	            IF #i_boFinishedOk OR #i_boErr THEN
	                #io_stTask1.bo_InProgress := FALSE;
	                #io_boAnyInProgress := FALSE;
	                #io_boEnable := FALSE;
	            END_IF;
	            
	        ELSIF #io_stTask2.bo_InProgress THEN
	            IF #i_boFinishedOk THEN
	                #io_stTask2.bo_FinishedOk := TRUE;
	            END_IF;
	            IF #i_boErr THEN
	                #io_stTask2.bo_FinishedError := TRUE;
	            END_IF;
	            
	            IF #i_boFinishedOk OR #i_boErr THEN
	                #io_stTask2.bo_InProgress := FALSE;
	                #io_boAnyInProgress := FALSE;
	                #io_boEnable := FALSE;
	            END_IF;
	            
	        ELSIF #io_stTask3.bo_InProgress THEN
	            IF #i_boFinishedOk THEN
	                #io_stTask3.bo_FinishedOk := TRUE;
	            END_IF;
	            IF #i_boErr THEN
	                #io_stTask3.bo_FinishedError := TRUE;
	            END_IF;
	            
	            IF #i_boFinishedOk OR #i_boErr THEN
	                #io_stTask3.bo_InProgress := FALSE;
	                #io_boAnyInProgress := FALSE;
	                #io_boEnable := FALSE;
	            END_IF;
	        END_IF;
	    END_IF;
	    
	    // 3. Запуск новой задачи из очереди (по приоритету 1 -> 2 -> 3)
	    IF NOT #io_boAnyInProgress AND NOT #io_boEnable THEN
	        IF #io_stTask1.bo_Trigger THEN
	            #io_iCmdInput := #io_stTask1.i_Code;
	            #io_stTask1.bo_InProgress := TRUE;
	            #io_boAnyInProgress := TRUE;
	            #io_boEnable := TRUE;
	            #io_stTask1.bo_Trigger := FALSE;
	            
	        ELSIF #io_stTask2.bo_Trigger THEN
	            #io_iCmdInput := #io_stTask2.i_Code;
	            #io_stTask2.bo_InProgress := TRUE;
	            #io_boAnyInProgress := TRUE;
	            #io_boEnable := TRUE;
	            #io_stTask2.bo_Trigger := FALSE;
	            
	        ELSIF #io_stTask3.bo_Trigger THEN
	            #io_iCmdInput := #io_stTask3.i_Code;
	            #io_stTask3.bo_InProgress := TRUE;
	            #io_boAnyInProgress := TRUE;
	            #io_boEnable := TRUE;
	            #io_stTask3.bo_Trigger := FALSE;
	        END_IF;
	    END_IF;
END_FUNCTION

FUNCTION_BLOCK "FB_Map_Siwarex_Core"
TITLE = Маппинг данных Siwarex CS
{ S7_Optimized_Access := 'FALSE' }
AUTHOR : S7C_Lib
FAMILY : Analog
VERSION : 1.4
// ==============================================================================
// Описание: Адаптированный маппинг из UDT_SIWA_CS. Обработка раздельных кодов 
//           ошибок (модуля и драйвера). Встроенный таймер Watchdog в STAT.
// ==============================================================================
   VAR 
      stat_Diag_CS_1 { ExternalAccessible := 'False'; ExternalVisible := 'False'; ExternalWritable := 'False'} : Struct   // Внутренняя память для Watchdog
         Old_Count { ExternalAccessible := 'False'; ExternalVisible := 'False'; ExternalWritable := 'False'} : Byte;
         Old_Weight { ExternalAccessible := 'False'; ExternalVisible := 'False'; ExternalWritable := 'False'} : Real;
         Last_Change_ms { ExternalAccessible := 'False'; ExternalVisible := 'False'; ExternalWritable := 'False'} : Real;
      END_STRUCT;
      stat_Diag_CS_2 { ExternalAccessible := 'False'; ExternalVisible := 'False'; ExternalWritable := 'False'} : Struct   // Внутренняя память для Watchdog
         Old_Count { ExternalAccessible := 'False'; ExternalVisible := 'False'; ExternalWritable := 'False'} : Byte;
         Old_Weight { ExternalAccessible := 'False'; ExternalVisible := 'False'; ExternalWritable := 'False'} : Real;
         Last_Change_ms { ExternalAccessible := 'False'; ExternalVisible := 'False'; ExternalWritable := 'False'} : Real;
      END_STRUCT;
   END_VAR

   VAR_TEMP 
      temp_Value_Changed : Bool;
      temp_Counter_Changed : Bool;
   END_VAR


BEGIN
	
	// ============================================================================
	// SCALE CS_1
	// ============================================================================
	
	// 1. Веса
	"DB_MAP".Scale_CS_1.Weight_Gross_kg := INT_TO_REAL("DB_SCALE_CS_1".s_PROCESS_VALUES.i_GROSS_WEIGHT_PROC);
	"DB_MAP".Scale_CS_1.Weight_Net_kg := INT_TO_REAL("DB_SCALE_CS_1".s_PROCESS_VALUES.i_NET_WEIGHT_PROC);
	"DB_MAP".Scale_CS_1.Weight_Tare_kg := INT_TO_REAL("DB_SCALE_CS_1".s_PROCESS_VALUES.i_TARE_WEIGHT_PROC);
	
	// 2. Статусы
	"DB_MAP".Scale_CS_1.Status.Standstill := "DB_SCALE_CS_1".s_PROCESS_VALUES.bo_STA_ST_STAND_SCALE_ON;
	"DB_MAP".Scale_CS_1.Status.Limit_1 := "DB_SCALE_CS_1".s_PROCESS_VALUES.bo_STA_LIMIT1_ON;
	"DB_MAP".Scale_CS_1.Status.Limit_2 := "DB_SCALE_CS_1".s_PROCESS_VALUES.bo_STA_LIMIT2_ON;
	"DB_MAP".Scale_CS_1.Status.Tared := "DB_SCALE_CS_1".s_PROCESS_VALUES.bo_STA_TARED;
	"DB_MAP".Scale_CS_1.Status.Quarter_D_Zero := "DB_SCALE_CS_1".s_PROCESS_VALUES.bo_STA_025_D_ZERO;
	"DB_MAP".Scale_CS_1.Status.Scale_Calibrated := "DB_SCALE_CS_1".s_PROCESS_VALUES.bo_STA_SCALE_CALIBRATED;
	"DB_MAP".Scale_CS_1.Status.Write_Protected := "DB_SCALE_CS_1".s_PROCESS_VALUES.bo_STA_WRI_PROT;
	"DB_MAP".Scale_CS_1.Status.Limit_Max := "DB_SCALE_CS_1".s_PROCESS_VALUES.bo_STA_MAX_9E;
	"DB_MAP".Scale_CS_1.Status.Fault_HW := "DB_SCALE_CS_1".s_PROCESS_VALUES.bo_STA_ERROR_ON;
	"DB_MAP".Scale_CS_1.Status.Fault_FB := "DB_SCALE_CS_1".bo_FB_ERR;
	"DB_MAP".Scale_CS_1.Status.Fault := "DB_SCALE_CS_1".s_PROCESS_VALUES.bo_STA_ERROR_ON OR "DB_SCALE_CS_1".bo_FB_ERR;
	
	// 3. Коды ошибок: старший байт = b_OPR_ERR_MSG, младший = b_FB_ERR_CODE
	"DB_MAP".Scale_CS_1.Err_Raw :=
	    SHL(IN := BYTE_TO_WORD("DB_SCALE_CS_1".s_PROCESS_VALUES.b_OPR_ERR_MSG), N := 8)
	    OR BYTE_TO_WORD("DB_SCALE_CS_1".b_FB_ERR_CODE);
	
	// 4. Watchdog CS_1
	#temp_Value_Changed := ("DB_MAP".Scale_CS_1.Weight_Net_kg <> #stat_Diag_CS_1.Old_Weight);
	#temp_Counter_Changed := ("DB_SCALE_CS_1".b_INFO_REFRESH_COUNT <> #stat_Diag_CS_1.Old_Count);
	
	IF #temp_Counter_Changed THEN //#temp_Value_Changed OR 
	    #stat_Diag_CS_1.Last_Change_ms := 0.0;
	    #stat_Diag_CS_1.Old_Weight := "DB_MAP".Scale_CS_1.Weight_Net_kg;
	    #stat_Diag_CS_1.Old_Count := "DB_SCALE_CS_1".b_INFO_REFRESH_COUNT;
	    "DB_MAP".Scale_CS_1.Status.Comm_Fault := FALSE;
	ELSE
	    #stat_Diag_CS_1.Last_Change_ms := #stat_Diag_CS_1.Last_Change_ms + "getCycleTime"();
	    IF #stat_Diag_CS_1.Last_Change_ms > 5000.0 THEN
	        "DB_MAP".Scale_CS_1.Status.Comm_Fault := TRUE;
	    END_IF;
	END_IF;
	
	
	// ============================================================================
	// SCALE CS_2
	// ============================================================================
	
	// 1. Веса
	"DB_MAP".Scale_CS_2.Weight_Gross_kg := INT_TO_REAL("DB_SCALE_CS_2".s_PROCESS_VALUES.i_GROSS_WEIGHT_PROC);
	"DB_MAP".Scale_CS_2.Weight_Net_kg := INT_TO_REAL("DB_SCALE_CS_2".s_PROCESS_VALUES.i_NET_WEIGHT_PROC);
	"DB_MAP".Scale_CS_2.Weight_Tare_kg := INT_TO_REAL("DB_SCALE_CS_2".s_PROCESS_VALUES.i_TARE_WEIGHT_PROC);
	
	// 2. Статусы
	"DB_MAP".Scale_CS_2.Status.Standstill := "DB_SCALE_CS_2".s_PROCESS_VALUES.bo_STA_ST_STAND_SCALE_ON;
	"DB_MAP".Scale_CS_2.Status.Limit_1 := "DB_SCALE_CS_2".s_PROCESS_VALUES.bo_STA_LIMIT1_ON;
	"DB_MAP".Scale_CS_2.Status.Limit_2 := "DB_SCALE_CS_2".s_PROCESS_VALUES.bo_STA_LIMIT2_ON;
	"DB_MAP".Scale_CS_2.Status.Tared := "DB_SCALE_CS_2".s_PROCESS_VALUES.bo_STA_TARED;
	"DB_MAP".Scale_CS_2.Status.Quarter_D_Zero := "DB_SCALE_CS_2".s_PROCESS_VALUES.bo_STA_025_D_ZERO;
	"DB_MAP".Scale_CS_2.Status.Scale_Calibrated := "DB_SCALE_CS_2".s_PROCESS_VALUES.bo_STA_SCALE_CALIBRATED;
	"DB_MAP".Scale_CS_2.Status.Write_Protected := "DB_SCALE_CS_2".s_PROCESS_VALUES.bo_STA_WRI_PROT;
	"DB_MAP".Scale_CS_2.Status.Limit_Max := "DB_SCALE_CS_2".s_PROCESS_VALUES.bo_STA_MAX_9E;
	"DB_MAP".Scale_CS_2.Status.Fault_HW := "DB_SCALE_CS_2".s_PROCESS_VALUES.bo_STA_ERROR_ON;
	"DB_MAP".Scale_CS_2.Status.Fault_FB := "DB_SCALE_CS_2".bo_FB_ERR;
	"DB_MAP".Scale_CS_2.Status.Fault := "DB_SCALE_CS_2".s_PROCESS_VALUES.bo_STA_ERROR_ON OR "DB_SCALE_CS_2".bo_FB_ERR;
	// 3. Коды ошибок
	"DB_MAP".Scale_CS_2.Err_Raw :=
	SHL(IN := BYTE_TO_WORD("DB_SCALE_CS_2".s_PROCESS_VALUES.b_OPR_ERR_MSG), N := 8)
	OR BYTE_TO_WORD("DB_SCALE_CS_2".b_FB_ERR_CODE);
	
	// 4. Watchdog CS_2
	#temp_Value_Changed := ("DB_MAP".Scale_CS_2.Weight_Net_kg <> #stat_Diag_CS_2.Old_Weight);
	#temp_Counter_Changed := ("DB_SCALE_CS_2".b_INFO_REFRESH_COUNT <> #stat_Diag_CS_2.Old_Count);
	
	IF #temp_Counter_Changed THEN //#temp_Value_Changed OR 
	    #stat_Diag_CS_2.Last_Change_ms := 0.0;
	    #stat_Diag_CS_2.Old_Weight := "DB_MAP".Scale_CS_2.Weight_Net_kg;
	    #stat_Diag_CS_2.Old_Count := "DB_SCALE_CS_2".b_INFO_REFRESH_COUNT;
	    "DB_MAP".Scale_CS_2.Status.Comm_Fault := FALSE;
	ELSE
	    #stat_Diag_CS_2.Last_Change_ms := #stat_Diag_CS_2.Last_Change_ms + "getCycleTime"();
	    IF #stat_Diag_CS_2.Last_Change_ms > 5000.0 THEN
	        "DB_MAP".Scale_CS_2.Status.Comm_Fault := TRUE;
	    END_IF;
	END_IF;
	
END_FUNCTION_BLOCK

FUNCTION "getCycleTime" : Real
{ S7_Optimized_Access := 'FALSE' }
VERSION : 0.1

BEGIN
	#getCycleTime := "DB_Global".Sys.CycleTime_ms_REAL;
END_FUNCTION

ORGANIZATION_BLOCK "COMPLETE RESTART"
TITLE = "Complete Restart"
{ S7_Optimized_Access := 'FALSE' }
VERSION : 0.1
   VAR_TEMP 
      OB100_EV_CLASS : Byte;   // 16#13, Event class 1, Entering event state, Event logged in diagnostic buffer
      OB100_STRTUP : Byte;   // 16#81/82/83/84 Method of startup
      OB100_PRIORITY : Byte;   // Priority of OB Execution
      OB100_OB_NUMBR : Byte;   // 100 (Organization block 100, OB100)
      OB100_RESERVED_1 : Byte;   // Reserved for system
      OB100_RESERVED_2 : Byte;   // Reserved for system
      OB100_STOP : Word;   // Event that caused CPU to stop (16#4xxx)
      OB100_STRT_INFO : DWord;   // Information on how system started
      OB100_DATE_TIME : Date_And_Time;   // Date and time OB100 started
   END_VAR


BEGIN
	"Total_DB".first_scan := TRUE;
	
END_ORGANIZATION_BLOCK

ORGANIZATION_BLOCK "CYC_INT5"
TITLE = "Cyclic Interrupt"
{ S7_Optimized_Access := 'FALSE' }
VERSION : 0.1
   VAR_TEMP 
      OB35_EV_CLASS : Byte;   // Bits 0-3 = 1 (Coming event), Bits 4-7 = 1 (Event class 1)
      OB35_STRT_INF : Byte;   // 16#36 (OB 35 has started)
      OB35_PRIORITY : Byte;   // Priority of OB Execution
      OB35_OB_NUMBR : Byte;   // 35 (Organization block 35, OB35)
      OB35_RESERVED_1 : Byte;   // Reserved for system
      OB35_RESERVED_2 : Byte;   // Reserved for system
      OB35_PHASE_OFFSET : Word;   // Phase offset (msec)
      OB35_RESERVED_3 : Int;   // Reserved for system
      OB35_EXC_FREQ : Int;   // Frequency of execution (msec)
      OB35_DATE_TIME : Date_And_Time;   // Date and time OB35 started
   END_VAR


BEGIN
	// Опрос Танка 1 (Слот 3 - фоновое чтение веса)
	"FC_Weighing_Poll"(
	                   i_boAnyInProgress := "DB_SCALE_CS_1".bo_CMD_IN_PROGRESS,
	                   i_boCmdEnable     := "DB_SCALE_CS_1".bo_CMD_TRIGGER,
	                   io_stTask          := "DB_SCALE_CS_1".s_CMD3
	);
	
	// Опрос Танка 2 (Слот 3 - фоновое чтение веса)
	"FC_Weighing_Poll"(
	                   i_boAnyInProgress := "DB_SCALE_CS_2".bo_CMD_IN_PROGRESS,
	                   i_boCmdEnable     := "DB_SCALE_CS_2".bo_CMD_TRIGGER,
	                   io_stTask          := "DB_SCALE_CS_2".s_CMD3
	);
END_ORGANIZATION_BLOCK

FUNCTION "FC_Weighing_Poll" : Void
{ S7_Optimized_Access := 'FALSE' }
VERSION : 1.2
   VAR_INPUT 
      i_boAnyInProgress : Bool;   // Общий статус занятости модуля
      i_boCmdEnable : Bool;   // Общий триггер команд модуля
   END_VAR

   VAR_IN_OUT 
      io_stTask : "UDT_SIWA_Cmd";   // Слот задачи циклического опроса (напр. sTask3)
   END_VAR


BEGIN
	    // ===================================================
	    // Генерация команды чтения Data Record (DR30 - Код 230)
	    // Функция предназначена для циклического вызова (OB35)
	    // ===================================================
	    IF NOT #i_boAnyInProgress AND NOT #i_boCmdEnable AND NOT #io_stTask.bo_InProgress THEN
	        #io_stTask.i_Code := 230;
	        #io_stTask.bo_Trigger := TRUE;
	    END_IF;
	    
END_FUNCTION

FUNCTION_BLOCK "FB_AI"
TITLE = Functional block from AI
{ S7_Optimized_Access := 'FALSE' }
AUTHOR : Gemini
FAMILY : Arhive
VERSION : 8.0
// -----------------------------------------------------------------------------
// БЛОК ОБРАБОТКИ АНАЛОГОВОГО СИГНАЛА (FB_AI)
// -----------------------------------------------------------------------------
   VAR_INPUT 
      i_iRawSignal : Int;
      i_rSimValue : Real;
   END_VAR

   VAR_IN_OUT 
      io_stConfig : "UDT_AI_Conf";
      io_stOut : "UDT_AI_Out";
   END_VAR

   VAR 
      stat_boWasInvalid : Bool := TRUE;
   END_VAR

   VAR_TEMP 
      temp_boDisabled : Bool;
      temp_boSimActive : Bool;
      temp_boUseSqrt : Bool;
      temp_boPreSqrtCut : Bool;
      temp_boFinalClamp : Bool;
      temp_rMA : Real;
      temp_rNorm : Real;
      temp_rCutoff_Norm : Real;
      temp_rScaled : Real;
      temp_rRange_mA : Real;
      temp_rRange_Phys : Real;
      temp_rMinPhys : Real;
      temp_rMaxPhys : Real;
      temp_boResetFilter : Bool;
      temp_iFilterTime : Int;
   END_VAR


BEGIN
	    // =========================================================
	    // ШАГ 0. РАСШИФРОВКА БИТОВОГО СЛОВА (Mode)
	    // =========================================================
	    #temp_boDisabled := (#io_stConfig.Mode AND 16#0001) = 16#0001;
	    #temp_boSimActive := (#io_stConfig.Mode AND 16#0002) = 16#0002;
	    #temp_boUseSqrt := (#io_stConfig.Mode AND 16#0004) = 16#0004;
	    #temp_boPreSqrtCut := (#io_stConfig.Mode AND 16#0008) = 16#0008;
	    #temp_boFinalClamp := (#io_stConfig.Mode AND 16#0010) = 16#0010;
	    
	    // 0.1 Режим полного отключения канала
	    IF #temp_boDisabled THEN
	        #io_stOut.Value_Unclamped := 0.0;
	        #io_stOut.Value_Scaled := 0.0;
	        #io_stOut.Value_Filtered := 0.0;
	        #io_stOut.Value_mA := 0.0;
	        #io_stOut.Raw := 0;
	        
	        #io_stOut.Status.WireBreak := FALSE;
	        #io_stOut.Status.Underrange := FALSE;
	        #io_stOut.Status.Overrange := FALSE;
	        #io_stOut.Status.Overflow := FALSE;
	        #io_stOut.Status.ConfigError := FALSE;
	        #io_stOut.Status.Sim_Active := FALSE;
	        
	        #stat_boWasInvalid := TRUE;
	        RETURN;
	    END_IF;
	    
	    // 0.2 Защита от ошибок конфигурации
	    #temp_rRange_mA := #io_stConfig.Calib_mA_Max - #io_stConfig.Calib_mA_Min;
	    #temp_rRange_Phys := #io_stConfig.Scale_Max - #io_stConfig.Scale_Min;
	    
	    IF (#io_stConfig.HW_Max <= #io_stConfig.HW_Min) OR
	        (#temp_rRange_mA <= 0.0) OR
	        (ABS(#temp_rRange_Phys) < 0.00001) OR
	        (ABS(#io_stConfig.Cutoff) >= ABS(#temp_rRange_Phys)) THEN
	        
	        #io_stOut.Status.ConfigError := TRUE;
	        
	        #io_stOut.Status.WireBreak := FALSE;
	        #io_stOut.Status.Underrange := FALSE;
	        #io_stOut.Status.Overrange := FALSE;
	        #io_stOut.Status.Overflow := FALSE;
	        #io_stOut.Status.Sim_Active := FALSE;
	        
	        #io_stOut.Value_Unclamped := 0.0;
	        #io_stOut.Value_Scaled := 0.0;
	        #io_stOut.Value_Filtered := 0.0;
	        #io_stOut.Value_mA := 0.0;
	        #io_stOut.Raw := #i_iRawSignal;
	        
	        #stat_boWasInvalid := TRUE;
	        RETURN;
	    END_IF;
	    
	    #io_stOut.Status.ConfigError := FALSE;
	    
	    // =========================================================
	    // ШАГ 1 & 2. СИМУЛЯЦИЯ И ДИАГНОСТИКА
	    // =========================================================
	    IF #temp_boSimActive THEN
	        #io_stOut.Status.Sim_Active := TRUE;
	        
	        #io_stOut.Status.WireBreak := FALSE;
	        #io_stOut.Status.Underrange := FALSE;
	        #io_stOut.Status.Overrange := FALSE;
	        #io_stOut.Status.Overflow := FALSE;
	        
	        #io_stOut.Raw := 0;
	        #io_stOut.Value_mA := 0.0;
	        #temp_rScaled := #i_rSimValue;
	    ELSE
	        #io_stOut.Status.Sim_Active := FALSE;
	        #io_stOut.Raw := #i_iRawSignal;
	        
	        "FC_AnalogDiag"(
	                        i_iRawSignal := #i_iRawSignal,
	                        i_iHW_Min := #io_stConfig.HW_Min,
	                        i_iHW_Max := #io_stConfig.HW_Max,
	                        i_rCoef_Under := "C_DIAG_UNDER",
	                        i_rCoef_Over := "C_DIAG_OVER",
	                        o_boWireBreak => #io_stOut.Status.WireBreak,
	                        o_boUnderrange => #io_stOut.Status.Underrange,
	                        o_boOverrange => #io_stOut.Status.Overrange,
	                        o_boOverflow => #io_stOut.Status.Overflow
	        );
	        
	        // =========================================================
	        // ШАГ 3. МАТЕМАТИКА
	        // =========================================================
	        IF #io_stOut.Status.WireBreak THEN
	            #temp_rScaled := #io_stConfig.Scale_Min + (#temp_rRange_Phys * "C_DIAG_UNDER");
	            #io_stOut.Value_mA := 0.0;
	            
	        ELSIF #io_stOut.Status.Overflow THEN
	            #temp_rScaled := #io_stConfig.Scale_Min + (#temp_rRange_Phys * "C_DIAG_OVER");
	            #io_stOut.Value_mA := 25.0;
	            
	        ELSE
	            // А) Расчет миллиампер
	            #temp_rMA := 4.0 + ((INT_TO_REAL(#i_iRawSignal) - INT_TO_REAL(#io_stConfig.HW_Min)) /
	            (INT_TO_REAL(#io_stConfig.HW_Max) - INT_TO_REAL(#io_stConfig.HW_Min))) * 16.0;
	            #io_stOut.Value_mA := #temp_rMA;
	            
	            // Б) Нормализация (0.0 ... 1.0)
	            #temp_rNorm := (#temp_rMA - #io_stConfig.Calib_mA_Min) / #temp_rRange_mA;
	            
	            // В & Г) Работа с корнем (Отсечка и извлечение)
	            IF #temp_boUseSqrt THEN
	                
	                IF #temp_boPreSqrtCut THEN
	                    #temp_rCutoff_Norm := #io_stConfig.Cutoff / #temp_rRange_Phys;
	                    #temp_rCutoff_Norm := #temp_rCutoff_Norm * #temp_rCutoff_Norm;
	                    
	                    IF #temp_rNorm < #temp_rCutoff_Norm THEN
	                        #temp_rNorm := 0.0;
	                    END_IF;
	                END_IF;
	                
	                IF #temp_rNorm > 0.0 THEN
	                    #temp_rNorm := SQRT(#temp_rNorm);
	                ELSE
	                    #temp_rNorm := 0.0;
	                END_IF;
	                
	            END_IF;
	            
	            // Д) Масштабирование в физическую величину
	            #temp_rScaled := #io_stConfig.Scale_Min + (#temp_rNorm * #temp_rRange_Phys);
	            
	            // Е) Классический CutOff (только если не применялся Pre-Sqrt)
	            IF NOT (#temp_boPreSqrtCut AND #temp_boUseSqrt) THEN
	                IF ABS(#temp_rScaled) < ABS(#io_stConfig.Cutoff) THEN
	                    #temp_rScaled := 0.0;
	                END_IF;
	            END_IF;
	        END_IF;
	    END_IF;
	    
	    // Сохраняем чистую математику на выход
	    #io_stOut.Value_Unclamped := #temp_rScaled;
	    
	    // =========================================================
	    // ШАГ 3.5. ФИНАЛЬНЫЙ CLAMP
	    // =========================================================
	    IF #temp_boFinalClamp THEN
	        #temp_rMinPhys := MIN(IN1 := #io_stConfig.Scale_Min, IN2 := #io_stConfig.Scale_Max);
	        #temp_rMaxPhys := MAX(IN1 := #io_stConfig.Scale_Min, IN2 := #io_stConfig.Scale_Max);
	        #temp_rScaled := LIMIT(MN := #temp_rMinPhys, IN := #temp_rScaled, MX := #temp_rMaxPhys);
	    END_IF;
	    
	    #io_stOut.Value_Scaled := #temp_rScaled;
	    
	    // =========================================================
	    // ШАГ 4. ФИЛЬТРАЦИЯ & PRE-LOAD 
	    // =========================================================
	    #temp_boResetFilter := #temp_boSimActive OR
	    #io_stOut.Status.WireBreak OR
	    #io_stOut.Status.Overflow OR
	    #stat_boWasInvalid;
	    
	    #temp_iFilterTime := LIMIT(MN := 0, IN := #io_stConfig.FilterTime_ms, MX := 32000);
	    
	    "FC_Filter_PT1"(
	                    i_rRawValue := #temp_rScaled,
	                    i_rTimeFilter_ms := INT_TO_REAL(#temp_iFilterTime),
	                    i_boReset := #temp_boResetFilter,
	                    io_rFilteredValue := #io_stOut.Value_Filtered
	    );
	    
	    #stat_boWasInvalid := #io_stOut.Status.WireBreak OR
	    #io_stOut.Status.Overflow OR
	    #io_stOut.Status.ConfigError;
	    
END_FUNCTION_BLOCK

FUNCTION "FC_AnalogDiag" : Void
{ S7_Optimized_Access := 'FALSE' }
VERSION : 1.1
   VAR_INPUT 
      i_iRawSignal : Int;
      i_iHW_Min : Int;
      i_iHW_Max : Int;
      i_rCoef_Under : Real;
      i_rCoef_Over : Real;
   END_VAR

   VAR_OUTPUT 
      o_boWireBreak : Bool;
      o_boUnderrange : Bool;
      o_boOverrange : Bool;
      o_boOverflow : Bool;
   END_VAR

   VAR_TEMP 
      temp_iLimit_Max : Real;
      temp_iLimit_Min : Int;
      temp_rHWRange : Real;
   END_VAR


BEGIN
	#temp_rHWRange := INT_TO_REAL(#i_iHW_Max) - INT_TO_REAL(#i_iHW_Min);
	
	#temp_iLimit_Max := REAL_TO_INT(INT_TO_REAL(#i_iHW_Max) + (#i_rCoef_Over * #temp_rHWRange));
	#temp_iLimit_Min := REAL_TO_INT(INT_TO_REAL(#i_iHW_Min) + (#i_rCoef_Under * #temp_rHWRange));
	
	#o_boWireBreak := #i_iRawSignal < #temp_iLimit_Min;
	#o_boUnderrange := (#i_iRawSignal < #i_iHW_Min) AND (#i_iRawSignal >= #temp_iLimit_Min);
	#o_boOverrange := (#i_iRawSignal > #i_iHW_Max) AND (#i_iRawSignal <= #temp_iLimit_Max);
	#o_boOverflow := #i_iRawSignal >#temp_iLimit_Max;
END_FUNCTION

FUNCTION "FC_Filter_PT1" : Void
{ S7_Optimized_Access := 'FALSE' }
VERSION : 1.3
// ==========================================
// МАТЕМАТИКА: ФИЛЬТР ЭКСПОНЕНЦИАЛЬНОГО СГЛАЖИВАНИЯ (PT1)
// ==========================================
   VAR_INPUT 
      i_rRawValue : Real;
      i_rTimeFilter_ms : Real;
      i_boReset : Bool;
   END_VAR

   VAR_IN_OUT 
      io_rFilteredValue : Real;
   END_VAR

   VAR_TEMP 
      temp_rCycleTime_ms : Real;
      temp_rAlpha : Real;
   END_VAR


BEGIN
	#temp_rCycleTime_ms := "getCycleTime"();
	
	//Защита
	// -Ресет фильтра
	// -Защита от системного сбоя (если ПЛК выдал dt <= 0)
	// -Умный Safe State (по правилу Найквиста)
	//    Если заданное время фильтра меньше половины цикла ПЛК,
	//    фильтрация физически невозможна. Просто пробрасываем сигнал напрямую.
	IF #i_boReset OR #temp_rCycleTime_ms <= 0.000001 OR #i_rTimeFilter_ms < (#temp_rCycleTime_ms / 2.0) THEN
	    #io_rFilteredValue := #i_rRawValue;
	    RETURN;
	END_IF;
	
	IF #i_rTimeFilter_ms < 50.0 THEN
	    #temp_rAlpha := 1.0;
	    #io_rFilteredValue := #i_rRawValue;
	    RETURN;
	END_IF;
	
	
	// 3. Математика PT1
	#temp_rAlpha := #temp_rCycleTime_ms / (#i_rTimeFilter_ms + #temp_rCycleTime_ms);
	#io_rFilteredValue := #io_rFilteredValue + #temp_rAlpha * (#i_rRawValue - #io_rFilteredValue);
	
END_FUNCTION

FUNCTION_BLOCK "FB_AI_Alarm"
{ S7_Optimized_Access := 'FALSE' }
VERSION : 2.0
   VAR_INPUT 
      i_rValue : Real;
      i_boReset : Bool;
      i_boInhibit : Bool;
   END_VAR

   VAR_IN_OUT 
      io_stConfig : "UDT_AI_Alarm_Conf";
      io_stOut : "UDT_AI_Alarm";
   END_VAR

   VAR 
      stat_TonHiHi {InstructionName := 'TON'; LibVersion := '1.0'; S7_SetPoint := 'False'} : TON;
      stat_TonHi {InstructionName := 'TON'; LibVersion := '1.0'; S7_SetPoint := 'False'} : TON;
      stat_TonLo {InstructionName := 'TON'; LibVersion := '1.0'; S7_SetPoint := 'False'} : TON;
      stat_TonLoLo {InstructionName := 'TON'; LibVersion := '1.0'; S7_SetPoint := 'False'} : TON;
      stat_RawHiHi : Bool;
      stat_RawHi : Bool;
      stat_RawLo : Bool;
      stat_RawLoLo : Bool;
   END_VAR


BEGIN
	    // =========================================================
	    // 0. ЗАЩИТА ОТ ДУРАКА (Ограничение уставок времени >= 0)
	    // =========================================================
	    IF #io_stConfig.Delay_HiHi < 0 THEN
	        #io_stConfig.Delay_HiHi := 0;
	    END_IF;
	    IF #io_stConfig.Delay_Hi < 0 THEN
	        #io_stConfig.Delay_Hi := 0;
	    END_IF;
	    IF #io_stConfig.Delay_Lo < 0 THEN
	        #io_stConfig.Delay_Lo := 0;
	    END_IF;
	    IF #io_stConfig.Delay_LoLo < 0 THEN
	        #io_stConfig.Delay_LoLo := 0;
	    END_IF;
	    
	    // =========================================================
	    // 1. ТРАНСЛЯЦИЯ СТАТУСОВ ДЛЯ HMI (En_Out)
	    // =========================================================
	    #io_stOut.En_HiHi := #io_stConfig.En_Alarm.HiHi AND NOT #i_boInhibit;
	    #io_stOut.En_Hi := #io_stConfig.En_Alarm.Hi AND NOT #i_boInhibit;
	    #io_stOut.En_Lo := #io_stConfig.En_Alarm.Lo AND NOT #i_boInhibit;
	    #io_stOut.En_LoLo := #io_stConfig.En_Alarm.LoLo AND NOT #i_boInhibit;
	    #io_stOut.En_Latch_Enable := #io_stConfig.En_Alarm.Latch_Enable;
	    
	    // =========================================================
	    // 2. ОБРАБОТКА СЫРЫХ АВАРИЙ С ГИСТЕРЕЗИСОМ (Deadband)
	    // =========================================================
	    // Верхние пороги (Срабатывание >, Сброс <)
	    IF #i_rValue > #io_stConfig.HiHi THEN
	        #stat_RawHiHi := TRUE;
	    ELSIF #i_rValue < (#io_stConfig.HiHi - #io_stConfig.Hysteresis) THEN
	        #stat_RawHiHi := FALSE;
	    END_IF;
	    
	    IF #i_rValue > #io_stConfig.Hi THEN
	        #stat_RawHi := TRUE;
	    ELSIF #i_rValue < (#io_stConfig.Hi - #io_stConfig.Hysteresis) THEN
	        #stat_RawHi := FALSE;
	    END_IF;
	    
	    // Нижние пороги (Срабатывание <, Сброс >)
	    IF #i_rValue < #io_stConfig.Lo THEN
	        #stat_RawLo := TRUE;
	    ELSIF #i_rValue > (#io_stConfig.Lo + #io_stConfig.Hysteresis) THEN
	        #stat_RawLo := FALSE;
	    END_IF;
	    
	    IF #i_rValue < #io_stConfig.LoLo THEN
	        #stat_RawLoLo := TRUE;
	    ELSIF #i_rValue > (#io_stConfig.LoLo + #io_stConfig.Hysteresis) THEN
	        #stat_RawLoLo := FALSE;
	    END_IF;
	    
	    // =========================================================
	    // 3. ТАЙМЕРЫ ЗАДЕРЖКИ (ON-Delay)
	    // =========================================================
	    // Таймер не считает, если сработала блокировка датчика (Inhibit) 
	    // или аларм выключен в настройках.
	    #stat_TonHiHi(IN := #stat_RawHiHi AND #io_stConfig.En_Alarm.HiHi AND NOT #i_boInhibit,
	                  PT := DINT_TO_TIME(#io_stConfig.Delay_HiHi) * 1000 + t#1ms);//gr-ny 300
	    
	    #stat_TonHi(IN := #stat_RawHi AND #io_stConfig.En_Alarm.Hi AND NOT #i_boInhibit,
	                PT := DINT_TO_TIME(#io_stConfig.Delay_Hi) * 1000 + t#1ms);//gr-ny 300
	    
	    #stat_TonLo(IN := #stat_RawLo AND #io_stConfig.En_Alarm.Lo AND NOT #i_boInhibit,
	                PT := DINT_TO_TIME(#io_stConfig.Delay_Lo) * 1000 + t#1ms);//gr-ny 300
	    
	    #stat_TonLoLo(IN := #stat_RawLoLo AND #io_stConfig.En_Alarm.LoLo AND NOT #i_boInhibit,
	                  PT := DINT_TO_TIME(#io_stConfig.Delay_LoLo) * 1000 + t#1ms);//gr-ny 300
	    
	    // =========================================================
	    // 4. ФИКСАЦИЯ (LATCH) И СБРОС АВАРИЙ
	    // =========================================================
	    // Логика сброса (имеет приоритет):
	    // 1. Сработал Inhibit (глушим всё безусловно)
	    // 2. Аларм сняли в настройках
	    // 3. Уровень в норме И (нет фиксации ИЛИ нажата кнопка Reset)
	    
	    // --- HiHi ---
	    IF #i_boInhibit OR NOT #io_stConfig.En_Alarm.HiHi OR
	        (NOT #stat_RawHiHi AND (NOT #io_stConfig.En_Alarm.Latch_Enable OR #i_boReset)) THEN
	        #io_stOut.HiHi := FALSE;
	    ELSIF #stat_TonHiHi.Q THEN
	        #io_stOut.HiHi := TRUE;
	    END_IF;
	    
	    // --- Hi ---
	    IF #i_boInhibit OR NOT #io_stConfig.En_Alarm.Hi OR
	        (NOT #stat_RawHi AND (NOT #io_stConfig.En_Alarm.Latch_Enable OR #i_boReset)) THEN
	        #io_stOut.Hi := FALSE;
	    ELSIF #stat_TonHi.Q THEN
	        #io_stOut.Hi := TRUE;
	    END_IF;
	    
	    // --- Lo ---
	    IF #i_boInhibit OR NOT #io_stConfig.En_Alarm.Lo OR
	        (NOT #stat_RawLo AND (NOT #io_stConfig.En_Alarm.Latch_Enable OR #i_boReset)) THEN
	        #io_stOut.Lo := FALSE;
	    ELSIF #stat_TonLo.Q THEN
	        #io_stOut.Lo := TRUE;
	    END_IF;
	    
	    // --- LoLo ---
	    IF #i_boInhibit OR NOT #io_stConfig.En_Alarm.LoLo OR
	        (NOT #stat_RawLoLo AND (NOT #io_stConfig.En_Alarm.Latch_Enable OR #i_boReset)) THEN
	        #io_stOut.LoLo := FALSE;
	    ELSIF #stat_TonLoLo.Q THEN
	        #io_stOut.LoLo := TRUE;
	    END_IF;
	    
END_FUNCTION_BLOCK

FUNCTION_BLOCK "FB_DI"
TITLE = Func Block from DI
{ S7_Optimized_Access := 'FALSE' }
VERSION : 1.2
// ==============================================================================
// Файл: S7C_FC_Filter_PT1.scl
// Целевые ПЛК: S7-1200 / S7-1500 (Линейка Current)
// Особенности: 
// - Оптимизированный доступ (Optimized block access = TRUE)
// - Использование современных системных функций (время цикла, первый скан)
// - Кодировка при сохранении: UTF-8 with BOM
// ==============================================================================
   VAR_INPUT 
      i_boRaw { ExternalAccessible := 'False'; ExternalVisible := 'False'; ExternalWritable := 'False'} : Bool;   // Сырой физический вход
   END_VAR

   VAR_IN_OUT 
      io_stConfig : "UDT_DI_Conf";
      io_stOut : "UDT_DI_Out";
   END_VAR

   VAR 
      stat_TonFlt {InstructionName := 'TON_TIME'; LibVersion := '1.0'; ExternalAccessible := 'False'; ExternalVisible := 'False'; ExternalWritable := 'False'; S7_SetPoint := 'False'} : TON_TIME;   // Задержка включения
      stat_TofFlt {InstructionName := 'TOF_TIME'; LibVersion := '1.0'; ExternalAccessible := 'False'; ExternalVisible := 'False'; ExternalWritable := 'False'; S7_SetPoint := 'False'} : TOF_TIME;   // Задержка выключения
      stat_Mode { ExternalAccessible := 'False'; ExternalVisible := 'False'; ExternalWritable := 'False'} : Int;   // Текущий рабочий режим
      stat_OldMode { ExternalAccessible := 'False'; ExternalVisible := 'False'; ExternalWritable := 'False'} : Int;   // Предыдущий режим для отслеживания изменений
   END_VAR

   VAR_TEMP 
      temp_FilterTime : Time;
      temp_boDisabled : Bool;
      temp_boNorm : Bool;
      temp_boInvert : Bool;
   END_VAR


BEGIN
	    
	    #temp_boDisabled := (#io_stConfig.Mode = "DB_Global".c_stDI_Mode.Disabled);
	    
	    IF #temp_boDisabled THEN
	        #stat_Mode := "DB_Global".c_stDI_Mode.None;
	        RETURN;
	    END_IF;
	    
	    // =========================================================
	    // 1. ПРОВЕРКА РЕЖИМА И ПРЕОБРАЗОВАНИЕ ВРЕМЕНИ
	    // =========================================================
	    #stat_Mode := #io_stConfig.Mode;
	    
	    IF #stat_Mode < 0 OR #stat_Mode > "DB_Global".c_stDI_Mode.Disabled THEN
	        #stat_Mode := "DB_Global".c_stDI_Mode.None;
	    END_IF;
	    
	    // Преобразуем мс (Int) в формат Time
	    #temp_FilterTime := DINT_TO_TIME(INT_TO_DINT(#io_stConfig.FilterTime));
	    
	    // =========================================================
	    // 2. СБРОС ТАЙМЕРОВ ПРИ СМЕНЕ РЕЖИМА
	    // =========================================================
	    IF #stat_Mode <> #stat_OldMode THEN
	        #stat_TonFlt(IN := FALSE,
	                     PT := #temp_FilterTime);
	        #stat_TofFlt(IN := FALSE,
	                     PT := #temp_FilterTime);
	        
	        #io_stOut.Value := #i_boRaw;
	        #stat_OldMode := #stat_Mode;
	    END_IF;
	    
	    // =========================================================
	    // 3. ЛОГИКА ФИЛЬТРАЦИИ И ИНВЕРСИИ
	    // =========================================================
	    IF #stat_Mode = "DB_Global".c_stDI_Mode.None THEN
	        // Режим 0: Прямая передача сигнала (без фильтра)
	        #io_stOut.Value := #i_boRaw;
	        
	        // Сбрасываем таймеры, чтобы они не висели в фоне
	        #stat_TonFlt(IN := FALSE,
	                     PT := #temp_FilterTime);
	        #stat_TofFlt(IN := FALSE,
	                     PT := #temp_FilterTime);
	        
	    ELSE
	        // Режимы с фильтром: применяем TON и TOF
	        #stat_TonFlt(IN := #i_boRaw,
	                     PT := #temp_FilterTime);
	        #stat_TofFlt(IN := #i_boRaw,
	                     PT := #temp_FilterTime);
	        
	        // Включение (TON отработал) -> сигнал стабильно TRUE
	        IF #stat_TonFlt.Q THEN
	            #io_stOut.Value := (#stat_Mode = "DB_Global".c_stDI_Mode.NOpen);
	        END_IF;
	        
	        // Выключение (TOF отработал) -> сигнал стабильно FALSE
	        IF NOT #stat_TofFlt.Q THEN
	            #io_stOut.Value := (#stat_Mode <> "DB_Global".c_stDI_Mode.NOpen); // Сбрасываем соответственно режиму
	        END_IF;
	    END_IF;
	    
END_FUNCTION_BLOCK

FUNCTION_BLOCK "FB_DI_Alarm"
{ S7_Optimized_Access := 'FALSE' }
VERSION : 1.0
// =============================================================================
// БЛОК ДИСКРЕТНОГО АЛАРМА
// =============================================================================
   VAR_INPUT 
      i_boSignal : Bool;   // Обработанный сигнал (от FB_DI)
      i_boReset : Bool;   // Команда сброса (Квитирование)
      i_boInhibit : Bool;   // Блокировка (например, при потере питания шкафа)
   END_VAR

   VAR_IN_OUT 
      io_stConfig : "UDT_DI_Alarm_Conf";
      io_stOut : "UDT_DI_Alarm";
   END_VAR

   VAR 
      stat_TonAlarm {InstructionName := 'TON'; LibVersion := '1.0'; S7_SetPoint := 'False'} : TON;   // Таймер задержки срабатывания
      stat_InputInv : Bool;   // Внутренний статус после учета инверсии
   END_VAR


BEGIN
	    // =========================================================
	    // 0. ЗАЩИТА ОТ ДУРАКА
	    // =========================================================
	    IF #io_stConfig.Delay < 0 THEN
	        #io_stConfig.Delay := 0;
	    END_IF;
	    
	    // =========================================================
	    // 1. ТРАНСЛЯЦИЯ СТАТУСОВ ДЛЯ HMI (En_Out)
	    // =========================================================
	    #io_stOut.En_Alarm := #io_stConfig.En_Alarm AND NOT #i_boInhibit;
	    #io_stOut.Latch_Enable := #io_stConfig.Latch_Enable;
	    #io_stOut.Input_Raw := #i_boSignal;
	    
	    // =========================================================
	    // 2. ИНВЕРСИЯ СИГНАЛА (XOR)
	    // =========================================================
	    // Если Invert=0: Авария наступает при Signal=TRUE (замыкание)
	    // Если Invert=1: Авария наступает при Signal=FALSE (размыкание)
	    #stat_InputInv := #i_boSignal XOR #io_stConfig.Invert;
	    #io_stOut.Input_Inv := #stat_InputInv;
	    
	    // =========================================================
	    // 3. ТАЙМЕР ЗАДЕРЖКИ (В СЕКУНДАХ)
	    // =========================================================
	    // Вычисляем время и передаем в таймер. Если Inhibit активен или аларм выключен - таймер сбрасывается.
	    #stat_TonAlarm(IN := #stat_InputInv AND #io_stOut.En_Alarm,
	                   PT := DINT_TO_TIME(INT_TO_DINT(#io_stConfig.Delay)) * 1000 + t#1ms);//gr-ny 300
	    
	    // =========================================================
	    // 4. ЛОГИКА ФИКСАЦИИ (LATCH) И СБРОСА
	    // =========================================================
	    // Сброс происходит, если:
	    // 1. Сработала внешняя блокировка (Inhibit)
	    // 2. Авария выключена в конфигурации
	    // 3. Сигнал в норме И (нет фиксации ИЛИ нажата кнопка сброса)
	    
	    IF #i_boInhibit OR NOT #io_stConfig.En_Alarm OR
	        (NOT #stat_InputInv AND (NOT #io_stConfig.Latch_Enable OR #i_boReset)) THEN
	        #io_stOut.Alarm := FALSE;
	    ELSIF #stat_TonAlarm.Q THEN
	        #io_stOut.Alarm := TRUE;
	    END_IF;
	    
END_FUNCTION_BLOCK

FUNCTION_BLOCK "FB_Time_Trigger"
TITLE = 'Генератор часовых слепков (Пуленепробиваемый)'
{ S7_Optimized_Access := 'FALSE' }
AUTHOR : S7A_Lib
FAMILY : Archive
VERSION : 1.1
   VAR_INPUT 
      i_Shift_1_Start { ExternalAccessible := 'False'; ExternalVisible := 'False'; ExternalWritable := 'False'} : Int := 8;   // Час начала дневной смены (напр. 08:00)
      i_Shift_2_Start { ExternalAccessible := 'False'; ExternalVisible := 'False'; ExternalWritable := 'False'} : Int := 20;   // Час начала ночной смены (напр. 20:00)
   END_VAR

   VAR_OUTPUT 
      q_Trigger_Hour { ExternalAccessible := 'False'; ExternalVisible := 'False'; ExternalWritable := 'False'} : Bool;   // Импульс: Сменился час (или день)
      q_Trigger_Shift { ExternalAccessible := 'False'; ExternalVisible := 'False'; ExternalWritable := 'False'} : Bool;   // Импульс: Началась новая смена
   END_VAR

   VAR 
      stat_Prev_Hour { ExternalAccessible := 'False'; ExternalVisible := 'False'; ExternalWritable := 'False'} : Int;
      stat_Prev_Day { ExternalAccessible := 'False'; ExternalVisible := 'False'; ExternalWritable := 'False'} : Int;   // ДОБАВЛЕНО: Память предыдущего дня
      stat_Init_Done { ExternalAccessible := 'False'; ExternalVisible := 'False'; ExternalWritable := 'False'} : Bool;
      temp_DT { ExternalAccessible := 'False'; ExternalVisible := 'False'; ExternalWritable := 'False'} : Date_And_Time;
      temp_DT_Bytes { ExternalAccessible := 'False'; ExternalVisible := 'False'; ExternalWritable := 'False'} AT temp_DT : Array[0..7] of Byte;
      temp_Second_Int { ExternalAccessible := 'False'; ExternalVisible := 'False'; ExternalWritable := 'False'} : Int;
      temp_Minute_Int { ExternalAccessible := 'False'; ExternalVisible := 'False'; ExternalWritable := 'False'} : Int;
      temp_Hour_Int { ExternalAccessible := 'False'; ExternalVisible := 'False'; ExternalWritable := 'False'} : Int;
      temp_Day_Int { ExternalAccessible := 'False'; ExternalVisible := 'False'; ExternalWritable := 'False'} : Int;   // ДОБАВЛЕНО: Текущий день
      temp_Month_Int { ExternalAccessible := 'False'; ExternalVisible := 'False'; ExternalWritable := 'False'} : Int;
      temp_Yar_Int { ExternalAccessible := 'False'; ExternalVisible := 'False'; ExternalWritable := 'False'} : Int;
      temp_RetVal { ExternalAccessible := 'False'; ExternalVisible := 'False'; ExternalWritable := 'False'} : Int;
   END_VAR


BEGIN
	    #q_Trigger_Hour := FALSE;
	    #q_Trigger_Shift := FALSE;
	    
	    #temp_RetVal := RD_SYS_T(OUT => #temp_DT);
	    
	    #temp_Second_Int := BCD16_TO_INT(BYTE_TO_WORD(#temp_DT_Bytes[5]));
	    #temp_Minute_Int := BCD16_TO_INT(BYTE_TO_WORD(#temp_DT_Bytes[4]));
	    #temp_Hour_Int := BCD16_TO_INT(BYTE_TO_WORD(#temp_DT_Bytes[3]));
	    
	    #temp_Day_Int := BCD16_TO_INT(BYTE_TO_WORD(#temp_DT_Bytes[2]));
	    #temp_Month_Int := BCD16_TO_INT(BYTE_TO_WORD(#temp_DT_Bytes[1]));
	    #temp_Yar_Int := BCD16_TO_INT(BYTE_TO_WORD(#temp_DT_Bytes[0]));
	    
	    "DB_DateTime".DT_Byte := #temp_DT_Bytes;
	    "DB_DateTime".DateTime_PLC := #temp_DT;
	    "DB_DateTime".Date_PLC := DT_TO_DATE(#temp_DT);
	    "DB_DateTime".TimeOfDay_PLC := DT_TO_TOD(#temp_DT);
	    
	    // Инициализация при первой заливке блока
	    IF NOT #stat_Init_Done THEN
	        #stat_Prev_Hour := #temp_Hour_Int;
	        #stat_Prev_Day := #temp_Day_Int;
	        #stat_Init_Done := TRUE;
	        #q_Trigger_Hour := TRUE;
	        RETURN;
	    END_IF;
	    
	    // Контроль смены часа ИЛИ смены дня (закрывает баг "ровно 24 часа")
	    IF (#temp_Hour_Int <> #stat_Prev_Hour) OR (#temp_Day_Int <> #stat_Prev_Day) THEN
	        
	        #q_Trigger_Hour := TRUE;
	        
	        // Проверяем на начало смены
	        IF (#temp_Hour_Int = #i_Shift_1_Start) OR (#temp_Hour_Int = #i_Shift_2_Start) THEN
	            #q_Trigger_Shift := TRUE;
	        END_IF;
	        
	        // Обновляем память
	        #stat_Prev_Hour := #temp_Hour_Int;
	        #stat_Prev_Day := #temp_Day_Int;
	        
	    END_IF;
	    
END_FUNCTION_BLOCK

FUNCTION "FC_ScaleValue" : Real
{ S7_Optimized_Access := 'FALSE' }
VERSION : 1.2
// ==========================================
// МАТЕМАТИКА: БЕЗОПАСНОЕ МАСШТАБИРОВАНИЕ
// ==========================================
   VAR_INPUT 
      i_rInp : Real;   // Входное сырое значение
      i_rInpLow : Real;   // Нижний предел входа (напр. 0.0)
      i_rInpHigh : Real;   // Верхний предел входа (напр. 27648.0)
      i_rOutLow : Real;   // Нижний предел шкалы датчика
      i_rOutHigh : Real;   // Верхний предел шкалы датчика
      i_boUseSqrt : Bool;   // Флаг извлечения корня (для перепада давления)
      i_rCutoff : Real;   // Порог отсечения микрошумов около нуля (Мертвая зона)
      i_boUseLimit : Bool;   // Флаг использования обрезки
   END_VAR

   VAR_TEMP 
      temp_rPerc : Real;   // Нормализованное значение (0.0 .. 1.0)
      temp_rResult : Real;   // Промежуточный результат
   END_VAR


BEGIN
	    // 1. Защита от деления на ноль при неверной конфигурации
	    IF ABS(#i_rInpHigh - #i_rInpLow) < 0.00001 THEN
	        #FC_ScaleValue := 0.0;
	        RETURN;
	    END_IF;
	    
	    // 2. Линейная нормализация
	    #temp_rPerc := (#i_rInp - #i_rInpLow) / (#i_rInpHigh - #i_rInpLow);
	    
	    // 3. Применение обрезки, если установлен флаг i_boUseLimit
	    IF #i_boUseLimit THEN
	        // Встроенная функция LIMIT жестко удерживает значение в рамках 0.0 .. 1.0
	        #temp_rPerc := LIMIT(MN := 0.0, IN := #temp_rPerc, MX := 1.0);
	    END_IF;
	    
	    // 4. Извлечение квадратного корня с защитой от отрицательных чисел
	    IF #i_boUseSqrt THEN
	        IF #temp_rPerc < 0.0 THEN
	            #temp_rPerc := 0.0;
	        END_IF;
	        #temp_rPerc := SQRT(#temp_rPerc);
	    END_IF;
	    
	    // 5. Масштабирование в выходной диапазон
	    #temp_rResult := #temp_rPerc * (#i_rOutHigh - #i_rOutLow) + #i_rOutLow;
	    
	    // 6. Мертвая зона с использованием модуля (ABS) для поддержки биполярных шкал
	    IF (ABS(#temp_rResult) < #i_rCutoff) AND (ABS(#i_rCutoff) > 0.001) THEN
	        #FC_ScaleValue := 0.0;
	    ELSE
	        #FC_ScaleValue := #temp_rResult;
	    END_IF;
	    
END_FUNCTION

FUNCTION "FC_Sys_Update" : Void
{ S7_Optimized_Access := 'FALSE' }
VERSION : 0.1
// 3. SYSTEM FUNCTIONS
   VAR_INPUT 
      i_Scan_1 : Byte;
      i_Prev_Cycle : Int;
   END_VAR

   VAR_TEMP 
      tmp_dint : DInt;
   END_VAR


BEGIN
	
	"DB_Global".Sys.FirstScan := (#i_Scan_1 = 16#01);
	"DB_Global".Sys.CycleTime_ms_INT := #i_Prev_Cycle;
	IF #i_Prev_Cycle <= 0 THEN
	    #tmp_dint := 1;
	ELSE
	    #tmp_dint := INT_TO_DINT(#i_Prev_Cycle);
	END_IF;
	"DB_Global".Sys.CycleTime_ms_REAL := DINT_TO_REAL(#tmp_dint);
	
END_FUNCTION

FUNCTION "Formula_weight_tank" : Void
{ S7_Optimized_Access := 'FALSE' }
VERSION : 0.1
   VAR_INPUT 
      S : Real;
      P : Real;
      Den : Real;
   END_VAR

   VAR_IN_OUT 
      P_z : Real;
      P_w : Real;
      Zero_But : Bool;
      Weight_But : Bool;
      Weight : Real;
      Weight_zero : Real;
      Weight_DB : Real;
      Korect : Bool;
   END_VAR


BEGIN
	#Weight := (#S * ((#P / (9.81 * #Den)) * 100)) * #Den;
	
	IF #Zero_But = TRUE
	THEN
	    #Weight_zero := #Weight;
	    #P_z := #P;
	    #Zero_But := FALSE;
	END_IF;
	
	IF #Weight_But = TRUE
	THEN
	    #Weight_DB := #Weight-#Weight_zero;
	    #P_w := #P;
	    #Weight_But := FALSE;
	END_IF;
	
	IF #Korect = TRUE
	THEN
	    #Weight_DB := (#S * (((#P_w - #P_z) / (9.81 * #Den)) * 100)) * #Den;
	    #Korect := FALSE;
	END_IF;
END_FUNCTION

FUNCTION_BLOCK "FB_Tank_Logic"
TITLE = Tank Coordinator
{ S7_Optimized_Access := 'FALSE' }
AUTHOR : Gemini
FAMILY : Archive
VERSION : 1.2
   VAR_INPUT 
      i_iRaw_AI : Int;   // Аналоговый вход (PIW)
      i_rRaw_Siwa : Real;   // Вес напрямую с Siwarex
      i_boRaw_DI : Bool;   // Дискретный датчик (ВУ)
   END_VAR

   VAR_IN_OUT 
      io_Tank : "UDT_Tank_Full";   // Твои блоки как мультиэкземпляры
   END_VAR

   VAR 
      stat_AI : "FB_AI";
      stat_AI_Alarm : "FB_AI_Alarm";
      stat_DI : "FB_DI";
      stat_DI_Alarm : "FB_DI_Alarm";
   END_VAR

   VAR_TEMP 
      temp_Tank : "UDT_Tank_Full";
      temp_rCalcInput : Real;
      temp_boIsSiwa : Bool;
      temp_boInhibitAI : Bool;
   END_VAR


BEGIN
	#temp_Tank := #io_Tank;
	(*
	// 0. ПРОВЕРКА НАЛИЧИЯ (Is_Present)
	// Если датчик не установлен в конфиге - не мучаем контроллер расчетами
	IF NOT #temp_Tank.DI_Conf.Is_Present AND NOT #temp_Tank.AI_Conf.Is_Present THEN
	    RETURN;
	END_IF;
	*)
	
	// 1. ОБРАБОТКА АНАЛОГОВОГО КАНАЛА
	// Вызываем твой блок масштабирования (всегда, т.к. там фильтрация)
	#stat_AI(i_iRawSignal := #i_iRaw_AI,
	         io_stConfig  := #temp_Tank.AI_Conf,
	         io_stOut     := #temp_Tank.AI_Out,
	         i_rSimValue  := 0.0);
	
	// Определяем источник (Бит 16#0020 в Mode)
	#temp_boIsSiwa := (#temp_Tank.AI_Conf.Mode AND 16#0020) = 16#0020;
	
	IF #temp_boIsSiwa THEN
	    #temp_rCalcInput := #i_rRaw_Siwa;
	ELSE
	    #temp_rCalcInput := #temp_Tank.AI_Out.Value_Filtered;
	END_IF;
	
	// 2. ВЫЗОВ МАТЕМАТИКИ
	"FC_Tank_Calc"(i_rValue  := #temp_rCalcInput,
	               i_boIsSiwa := #temp_boIsSiwa,
	               io_Geom   := #temp_Tank.Geom,
	               iq_Calc   := #temp_Tank.Calc);
	
	// 3. АВАРИИ ПО УРОВНЮ (AI)
	// Глушим алармы AI при аппаратных ошибках (Inhibit)
	#temp_boInhibitAI := #temp_Tank.AI_Out.Status.WireBreak OR
	#temp_Tank.AI_Out.Status.Overflow OR
	#temp_Tank.AI_Out.Status.ConfigError;
	
	#stat_AI_Alarm(i_rValue    := #temp_Tank.AI_Out.Value_Filtered, // Алармы всегда по %
	               i_boReset   := #temp_Tank.Cmd.ResetError,
	               i_boInhibit := #temp_boInhibitAI,
	               io_stConfig := #temp_Tank.AI_Alarm_Conf,
	               io_stOut    := #temp_Tank.AI_Alarm);
	
	// 4. ОБРАБОТКА ДАТЧИКА ВЕРХНЕГО УРОВНЯ (DI)
	// Чистим дребезг
	#stat_DI(i_boRaw     := #i_boRaw_DI,
	         io_stConfig := #temp_Tank.DI_Conf,
	         io_stOut    := #temp_Tank.DI_Out);
	
	// Логика аварии ВУ (независима от AI)
	#stat_DI_Alarm(i_boSignal  := #temp_Tank.DI_Out.Value,
	               i_boReset   := #temp_Tank.Cmd.ResetError,
	               i_boInhibit := FALSE,//temp_Tank.DI_Alarm_Conf.Inhibit_Manual,
	               io_stConfig := #temp_Tank.DI_Alarm_Conf,
	               io_stOut    := #temp_Tank.DI_Alarm);
	
	#io_Tank := #temp_Tank;
	
END_FUNCTION_BLOCK

FUNCTION "FC_Tank_Calc" : Void
TITLE = Tank Physics Calculator
{ S7_Optimized_Access := 'FALSE' }
AUTHOR : Gemini
FAMILY : Archive
VERSION : 1.2
// ==============================================================================
// Описание: Расчет физических показателей танка (Цилиндр).
//           Поддерживает режим весов (кг) и режим уровня (м).
// ==============================================================================
   VAR_INPUT 
      i_rValue : Real;   // Входящее значение (м или кг)
      i_boIsSiwa : Bool;   // TRUE = Весы (кг), FALSE = Уровень (м)
   END_VAR

   VAR_IN_OUT 
      io_Geom : "UDT_Tank_Geom";
      iq_Calc : "UDT_Tank_Calc";
   END_VAR

   VAR_TEMP 
      temp_rPI : Real;
      temp_rArea : Real;
      temp_rDensity : Real;
   END_VAR


BEGIN
	    // Константы и проверки безопасности
	    #temp_rPI := 3.141593;
	    
	    // Плотность не может быть 0 (защита от деления)
	    IF #io_Geom.Density_tm3 < 0.001 THEN
	        #temp_rDensity := 1.0;
	    ELSE
	        #temp_rDensity := #io_Geom.Density_tm3;
	    END_IF;
	    
	    // 1. Расчет площади основания (S = PI * R^2) и макс. объема
	    #temp_rArea := #temp_rPI * #io_Geom.Radius_m * #io_Geom.Radius_m;
	    #iq_Calc.Max_Volume_m3 := #temp_rArea * #io_Geom.Height_Full_m;
	    
	    // Проверка на корректность геометрии
	    IF #iq_Calc.Max_Volume_m3 < 0.01 OR #io_Geom.Height_Full_m < 0.01 THEN
	        RETURN; // Выходим, если танк "пустой" в настройках
	    END_IF;
	    
	    // 2. Основной расчет в зависимости от режима
	    IF #i_boIsSiwa THEN
	        // --- РЕЖИМ ВЕСОВ (Вход в кг) ---
	        #iq_Calc.Weight_t := #i_rValue / 1000.0;
	        #iq_Calc.Volume_m3 := #iq_Calc.Weight_t / #temp_rDensity; // V(м3) = m(т) / rho(т/м3) 
	        
	        // Уровень вычисляем обратно из объема
	        #iq_Calc.Level_m := #iq_Calc.Volume_m3 / #temp_rArea;
	    ELSE
	        // --- РЕЖИМ УРОВНЯ (Вход в м) ---
	        #iq_Calc.Level_m := #i_rValue / #temp_rDensity + #io_Geom.Sensor_Offset_m;
	        #iq_Calc.Volume_m3 := #iq_Calc.Level_m * #temp_rArea;
	        
	        // Вес вычисляем из объема
	        #iq_Calc.Weight_t := #iq_Calc.Volume_m3 * #temp_rDensity; // m(т) = V(м3) * rho(т/м3)
	    END_IF;
	    
	    // 3. Расчет процентов
	    #iq_Calc.Level_Pct := (#iq_Calc.Level_m / #io_Geom.Height_Full_m) * 100.0;
	    #iq_Calc.Volume_Pct := (#iq_Calc.Volume_m3 / #iq_Calc.Max_Volume_m3) * 100.0;
END_FUNCTION

FUNCTION "FC_Calc_Whause" : Void
{ S7_Optimized_Access := 'FALSE' }
VERSION : 0.1
   VAR_TEMP 
      temp_i : Int;
   END_VAR


BEGIN
	// ==============================================================================
	// СКЛАД TRN (3 танка)
	// ==============================================================================
	
	"DB_MAP".HMI_Whouse_TRN.Total_Volume_m3 := 0.0;
	"DB_MAP".HMI_Whouse_TRN.Total_Weight_t := 0.0;
	"DB_MAP".HMI_Whouse_TRN.Total_Ullage_pct := 0.0;
	"DB_MAP".HMI_Whouse_TRN.Total_Ullage_m3 := 0.0;
	"DB_MAP".HMI_Whouse_TRN.Tanks_In_Alarm := 0;
	
	FOR #temp_i := 1 TO "c_Count_TRN" DO
	    "FC_Wh_Totals_Aggregation"(io_Tanks := "DB_Wh_TRN".Tank[#temp_i],
	                               io_Whouse := "DB_MAP".HMI_Whouse_TRN);
	END_FOR;
	
	IF ("DB_MAP".HMI_Whouse_TRN.Total_Volume_m3 + "DB_MAP".HMI_Whouse_TRN.Total_Ullage_m3) >= 0.001 THEN
	    "DB_MAP".HMI_Whouse_TRN.Total_Ullage_pct :=
	    "DB_MAP".HMI_Whouse_TRN.Total_Ullage_m3 / ("DB_MAP".HMI_Whouse_TRN.Total_Volume_m3 + "DB_MAP".HMI_Whouse_TRN.Total_Ullage_m3) * 100.0;
	END_IF;
	
	"DB_MAP".HMI_Whouse_TRN.Status_Word.Global_Alarm := ("DB_MAP".HMI_Whouse_TRN.Tanks_In_Alarm > 0);
	
	// Сброс глобальной кнопки после прохода цикла
	IF "DB_MAP".HMI_Whouse_TRN.Cmd_Word.Reset_All THEN
	    "DB_MAP".HMI_Whouse_TRN.Cmd_Word.Reset_All := FALSE;
	END_IF;
	
	// ==============================================================================
	// СКЛАД POL (10 танков)
	// ==============================================================================
	"DB_MAP".HMI_Whouse_POL.Total_Volume_m3 := 0.0;
	"DB_MAP".HMI_Whouse_POL.Total_Weight_t := 0.0;
	"DB_MAP".HMI_Whouse_POL.Total_Ullage_pct := 0.0;
	"DB_MAP".HMI_Whouse_POL.Total_Ullage_m3 := 0.0;
	"DB_MAP".HMI_Whouse_POL.Tanks_In_Alarm := 0;
	
	FOR #temp_i := 1 TO "c_Count_POL" DO
	    "FC_Wh_Totals_Aggregation"(io_Tanks := "DB_Wh_POL".Tank[#temp_i],
	                               io_Whouse := "DB_MAP".HMI_Whouse_POL);
	END_FOR;
	
	IF ("DB_MAP".HMI_Whouse_POL.Total_Volume_m3 + "DB_MAP".HMI_Whouse_POL.Total_Ullage_m3) >= 0.001 THEN
	    "DB_MAP".HMI_Whouse_POL.Total_Ullage_pct :=
	    "DB_MAP".HMI_Whouse_POL.Total_Ullage_m3 / ("DB_MAP".HMI_Whouse_POL.Total_Volume_m3 + "DB_MAP".HMI_Whouse_POL.Total_Ullage_m3) * 100.0;
	END_IF;
	"DB_MAP".HMI_Whouse_POL.Status_Word.Global_Alarm := ("DB_MAP".HMI_Whouse_POL.Tanks_In_Alarm > 0);
	
	// Сброс глобальной кнопки после прохода цикла
	IF "DB_MAP".HMI_Whouse_POL.Cmd_Word.Reset_All THEN
	    "DB_MAP".HMI_Whouse_POL.Cmd_Word.Reset_All := FALSE;
	END_IF;
	
	// ==============================================================================
	// СКЛАД BUL (4 танка)
	// ==============================================================================
	"DB_MAP".HMI_Whouse_BUL.Total_Volume_m3 := 0.0;
	"DB_MAP".HMI_Whouse_BUL.Total_Weight_t := 0.0;
	"DB_MAP".HMI_Whouse_BUL.Total_Ullage_pct := 0.0;
	"DB_MAP".HMI_Whouse_BUL.Total_Ullage_m3 := 0.0;
	"DB_MAP".HMI_Whouse_BUL.Tanks_In_Alarm := 0;
	
	FOR #temp_i := 1 TO "c_Count_BUL" DO
	    "FC_Wh_Totals_Aggregation"(io_Tanks := "DB_Wh_BUL".Tank[#temp_i],
	                               io_Whouse := "DB_MAP".HMI_Whouse_BUL);
	END_FOR;
	
	IF ("DB_MAP".HMI_Whouse_BUL.Total_Volume_m3 + "DB_MAP".HMI_Whouse_BUL.Total_Ullage_m3) >= 0.001 THEN
	    "DB_MAP".HMI_Whouse_BUL.Total_Ullage_pct :=
	    "DB_MAP".HMI_Whouse_BUL.Total_Ullage_m3 / ("DB_MAP".HMI_Whouse_BUL.Total_Volume_m3 + "DB_MAP".HMI_Whouse_BUL.Total_Ullage_m3) * 100.0;
	END_IF;
	
	"DB_MAP".HMI_Whouse_BUL.Status_Word.Global_Alarm := ("DB_MAP".HMI_Whouse_BUL.Tanks_In_Alarm > 0);
	
	// Сброс глобальной кнопки после прохода цикла
	IF "DB_MAP".HMI_Whouse_BUL.Cmd_Word.Reset_All THEN
	    "DB_MAP".HMI_Whouse_BUL.Cmd_Word.Reset_All := FALSE;
	END_IF;
	
	// ==============================================================================
	// СКЛАД MOL (12 танков)
	// ==============================================================================
	"DB_MAP".HMI_Whouse_MOL.Total_Volume_m3 := 0.0;
	"DB_MAP".HMI_Whouse_MOL.Total_Weight_t := 0.0;
	"DB_MAP".HMI_Whouse_MOL.Total_Ullage_pct := 0.0;
	"DB_MAP".HMI_Whouse_MOL.Total_Ullage_m3 := 0.0;
	"DB_MAP".HMI_Whouse_MOL.Tanks_In_Alarm := 0;
	
	FOR #temp_i := 1 TO "c_Count_MOL" DO
	    "FC_Wh_Totals_Aggregation"(io_Tanks := "DB_Wh_MOL".Tank[#temp_i],
	                               io_Whouse := "DB_MAP".HMI_Whouse_MOL);
	END_FOR;
	
	IF ("DB_MAP".HMI_Whouse_MOL.Total_Volume_m3 + "DB_MAP".HMI_Whouse_MOL.Total_Ullage_m3) >= 0.001 THEN
	    "DB_MAP".HMI_Whouse_MOL.Total_Ullage_pct :=
	    "DB_MAP".HMI_Whouse_MOL.Total_Ullage_m3 / ("DB_MAP".HMI_Whouse_MOL.Total_Volume_m3 + "DB_MAP".HMI_Whouse_MOL.Total_Ullage_m3) * 100.0;
	END_IF;
	
	"DB_MAP".HMI_Whouse_MOL.Status_Word.Global_Alarm := ("DB_MAP".HMI_Whouse_MOL.Tanks_In_Alarm > 0);
	
	// Сброс глобальной кнопки после прохода цикла
	IF "DB_MAP".HMI_Whouse_MOL.Cmd_Word.Reset_All THEN
	    "DB_MAP".HMI_Whouse_MOL.Cmd_Word.Reset_All := FALSE;
	END_IF;
	
	
END_FUNCTION

FUNCTION "FC_Wh_Totals_Aggregation" : Void
{ S7_Optimized_Access := 'FALSE' }
VERSION : 0.1
   VAR_IN_OUT 
      io_Tanks : "UDT_Tank_Full";
      io_Whouse : "UDT_HMI_Whouse";
   END_VAR

   VAR_TEMP 
      temp_AnyAlarm : Bool;
   END_VAR


BEGIN
	        // Агрегация объемов и весов
	        #io_Whouse.Total_Volume_m3 := #io_Whouse.Total_Volume_m3 + #io_Tanks.Calc.Volume_m3;
	        #io_Whouse.Total_Weight_t := #io_Whouse.Total_Weight_t + #io_Tanks.Calc.Weight_t;
	        #io_Whouse.Total_Ullage_m3 := #io_Whouse.Total_Ullage_m3 + (#io_Tanks.Calc.Max_Volume_m3 - #io_Tanks.Calc.Volume_m3);
	        
	        // Проверка наличия аварий в танке (HH, H, L, LL или DI) 
	        IF #io_Tanks.AI_Alarm.HiHi OR
	            #io_Tanks.AI_Alarm.Hi OR
	            #io_Tanks.AI_Alarm.Lo OR
	            #io_Tanks.AI_Alarm.LoLo OR
	            #io_Tanks.DI_Alarm.Alarm
	        THEN
	            #io_Whouse.Tanks_In_Alarm := #io_Whouse.Tanks_In_Alarm + 1;
	        END_IF;
	        
	        // Трансляция глобальной команды "Сброс всех аварий" [cite: 56, 82]
	        IF #io_Whouse.Cmd_Reset_All THEN
	            #io_Tanks.Cmd.ResetError := TRUE;
	        END_IF;
END_FUNCTION

FUNCTION "FC_Log_Mng" : Void
{ S7_Optimized_Access := 'FALSE' }
VERSION : 0.1
   VAR_TEMP 
      temp_Ind : Int;
   END_VAR


BEGIN
	
	
	FOR #temp_Ind := 1 TO "c_Count_TRN" DO
	    "FC_Log_Tank"(i_Whouse_ID:=1,
	                  i_Tank_Index:=INT_TO_BYTE(#temp_Ind),
	              io_Tank:="DB_HMI_MAP".TRN_SmalTank[#temp_Ind]);
	END_FOR;
	
	FOR #temp_Ind := 1 TO "c_Count_POL" DO
	    "FC_Log_Tank"(i_Whouse_ID := 2,
	                  i_Tank_Index := INT_TO_BYTE(#temp_Ind),
	                  io_Tank := "DB_HMI_MAP".POL_SmalTank[#temp_Ind]);
	END_FOR;
	
	FOR #temp_Ind := 1 TO "c_Count_BUL" DO
	    "FC_Log_Tank"(i_Whouse_ID := 3,
	                  i_Tank_Index := INT_TO_BYTE(#temp_Ind),
	                  io_Tank := "DB_HMI_MAP".BUL_SmalTank[#temp_Ind]);
	END_FOR;
	
	FOR #temp_Ind := 1 TO "c_Count_MOL" DO
	    "FC_Log_Tank"(i_Whouse_ID := 4,
	                  i_Tank_Index := INT_TO_BYTE(#temp_Ind),
	                  io_Tank := "DB_HMI_MAP".MOL_SmalTank[#temp_Ind]);
	END_FOR;
	
END_FUNCTION

FUNCTION "FC_Log_Tank" : Void
{ S7_Optimized_Access := 'FALSE' }
VERSION : 0.1
   VAR_INPUT 
      i_Whouse_ID : Byte;
      i_Tank_Index : Byte;
   END_VAR

   VAR_IN_OUT 
      io_Tank : "UDT_HMI_SmallTank";
   END_VAR

   VAR_TEMP 
      temp_Write_Ptr : Int;
      temp_DT : Date_And_Time;
   END_VAR


BEGIN
	
	#temp_DT := "DB_DateTime".DateTime_PLC;
	#temp_Write_Ptr := "DB_Log_Buffer".Write_Index;
	
	"DB_Log_Buffer".Buffer[#temp_Write_Ptr].Timestamp := #temp_DT;
	"DB_Log_Buffer".Buffer[#temp_Write_Ptr].Whouse_ID := #i_Whouse_ID;
	"DB_Log_Buffer".Buffer[#temp_Write_Ptr].Tank_Index := #i_Tank_Index;
	"DB_Log_Buffer".Buffer[#temp_Write_Ptr].Level_m := #io_Tank.Level_m;
	"DB_Log_Buffer".Buffer[#temp_Write_Ptr].Weight_t := #io_Tank.Weight_t;
	//"DB_Log_Buffer".Buffer[#temp_Write_Ptr].Status_Bits := #temp_Status;
	
	#temp_Write_Ptr := #temp_Write_Ptr + 1;
	IF #temp_Write_Ptr > 1999 THEN
	    #temp_Write_Ptr := 0;
	END_IF;
END_FUNCTION

FUNCTION "FC_Map_SmallTank_HMI" : Void
TITLE = Маппинг HMI малого танка
{ S7_Optimized_Access := 'FALSE' }
AUTHOR : S7A_Lib
FAMILY : HMI_Map
VERSION : 0.1
// ==============================================================================
// Описание: Перекладывает данные из внутренней структуры малого танка 
//           в плоскую HMI-структуру. Включает конвертацию массы в тонны 
//           и сквозную передачу статусных битов.
// ==============================================================================
   VAR_INPUT 
      i_Tank_Internal : "UDT_Tank_Full";   // Рабочая (внутренняя) структура танка
   END_VAR

   VAR_IN_OUT 
      io_HMI_Tank : "UDT_HMI_SmallTank";   // Плоская структура для панели оператора
   END_VAR


BEGIN
	    // Перенос основных технологических параметров
	    #io_HMI_Tank.Level_m := #i_Tank_Internal.Calc.Level_m;
	    #io_HMI_Tank.Volume_m3 := #i_Tank_Internal.Calc.Volume_m3;
	    #io_HMI_Tank.Percent_prc := #i_Tank_Internal.Calc.Level_Pct;
	    
	    // UPDATE: Конвертация массы из килограммов в тонны для отображения оператору
	    #io_HMI_Tank.Weight_t := #i_Tank_Internal.Calc.Weight_t;
	    
	    // Маппинг статусных битов аварий (побитово)
	    #io_HMI_Tank.Status_Alarms.DI := #i_Tank_Internal.DI_Alarm.Alarm;
	    #io_HMI_Tank.Status_Alarms.HH := #i_Tank_Internal.AI_Alarm.HiHi;
	    #io_HMI_Tank.Status_Alarms.H := #i_Tank_Internal.AI_Alarm.Hi;
	    #io_HMI_Tank.Status_Alarms.L := #i_Tank_Internal.AI_Alarm.Lo;
	    #io_HMI_Tank.Status_Alarms.LL := #i_Tank_Internal.AI_Alarm.LoLo;
	    
	    // Маппинг аппаратной диагностики AI (побитово)
	    #io_HMI_Tank.Status_AI.WireBreak := #i_Tank_Internal.AI_Out.Status.WireBreak;
	    #io_HMI_Tank.Status_AI.Underrange := #i_Tank_Internal.AI_Out.Status.Underrange;
	    #io_HMI_Tank.Status_AI.Overrange := #i_Tank_Internal.AI_Out.Status.Overrange;
	    #io_HMI_Tank.Status_AI.Overflow := #i_Tank_Internal.AI_Out.Status.Overflow;
	    #io_HMI_Tank.Status_AI.ConfigError := #i_Tank_Internal.AI_Out.Status.ConfigError;
	    
END_FUNCTION

FUNCTION "FC_Wh_BUL_Mng" : Void
{ S7_Optimized_Access := 'FALSE' }
VERSION : 0.1
   VAR_TEMP 
      temp_Ind : Int;
   END_VAR


BEGIN
	// ---------------------------------------------------------------
	// Склад: Болгарский (BUL) — 4 бака
	// ---------------------------------------------------------------
	
	"iDB_BUL_Tank_Log_1"(i_iRaw_AI  := "DB_IO_MAP".AI_BUL_Tank_1,
	                     i_rRaw_Siwa := 0.0,
	                     i_boRaw_DI  := "DB_IO_MAP".DI_BUL_Tank_1,
	                     io_Tank     := "DB_Wh_BUL".Tank[1]);
	
	"iDB_BUL_Tank_Log_2"(i_iRaw_AI  := "DB_IO_MAP".AI_BUL_Tank_2,
	                     i_rRaw_Siwa := 0.0,
	                     i_boRaw_DI  := "DB_IO_MAP".DI_BUL_Tank_2,
	                     io_Tank     := "DB_Wh_BUL".Tank[2]);
	
	"iDB_BUL_Tank_Log_3"(i_iRaw_AI  := "DB_IO_MAP".AI_BUL_Tank_3,
	                     i_rRaw_Siwa := 0.0,
	                     i_boRaw_DI  := "DB_IO_MAP".DI_BUL_Tank_3,
	                     io_Tank     := "DB_Wh_BUL".Tank[3]);
	
	"iDB_BUL_Tank_Log_4"(i_iRaw_AI  := "DB_IO_MAP".AI_BUL_Tank_4,
	                     i_rRaw_Siwa := 0.0,
	                     i_boRaw_DI  := "DB_IO_MAP".DI_BUL_Tank_4,
	                     io_Tank     := "DB_Wh_BUL".Tank[4]);
	
	// HMI маппинг
	FOR #temp_Ind := 1 TO 4 DO
	    "FC_Map_SmallTank_HMI"(i_Tank_Internal := "DB_Wh_BUL".Tank[#temp_Ind],
	                           io_HMI_Tank     := "DB_MAP".HMI_BUL_SmalTank[#temp_Ind]);
	END_FOR;
	
END_FUNCTION

FUNCTION "FC_Wh_MOL_Mng" : Void
{ S7_Optimized_Access := 'FALSE' }
VERSION : 0.1
   VAR_TEMP 
      temp_Ind : Int;
   END_VAR


BEGIN
	// ---------------------------------------------------------------
	// Склад: МОЛОЧНЫЕ (MOL) — 12 баков
	// ---------------------------------------------------------------
	
	"iDB_MOL_Tank_Log_1"(i_iRaw_AI  := "DB_IO_MAP".AI_MOL_Tank_1,
	                     i_rRaw_Siwa := 0.0,
	                     i_boRaw_DI  := "DB_IO_MAP".DI_MOL_Tank_1,
	                     io_Tank     := "DB_Wh_MOL".Tank[1]);
	
	"iDB_MOL_Tank_Log_2"(i_iRaw_AI  := "DB_IO_MAP".AI_MOL_Tank_2,
	                     i_rRaw_Siwa := 0.0,
	                     i_boRaw_DI  := "DB_IO_MAP".DI_MOL_Tank_2,
	                     io_Tank     := "DB_Wh_MOL".Tank[2]);
	
	"iDB_MOL_Tank_Log_3"(i_iRaw_AI  := "DB_IO_MAP".AI_MOL_Tank_3,
	                     i_rRaw_Siwa := 0.0,
	                     i_boRaw_DI  := "DB_IO_MAP".DI_MOL_Tank_3,
	                     io_Tank     := "DB_Wh_MOL".Tank[3]);
	
	"iDB_MOL_Tank_Log_4"(i_iRaw_AI  := "DB_IO_MAP".AI_MOL_Tank_4,
	                     i_rRaw_Siwa := 0.0,
	                     i_boRaw_DI  := "DB_IO_MAP".DI_MOL_Tank_4,
	                     io_Tank     := "DB_Wh_MOL".Tank[4]);
	
	"iDB_MOL_Tank_Log_5"(i_iRaw_AI  := "DB_IO_MAP".AI_MOL_Tank_5,
	                     i_rRaw_Siwa := 0.0,
	                     i_boRaw_DI  := "DB_IO_MAP".DI_MOL_Tank_5,
	                     io_Tank     := "DB_Wh_MOL".Tank[5]);
	
	"iDB_MOL_Tank_Log_6"(i_iRaw_AI  := "DB_IO_MAP".AI_MOL_Tank_6,
	                     i_rRaw_Siwa := 0.0,
	                     i_boRaw_DI  := "DB_IO_MAP".DI_MOL_Tank_6,
	                     io_Tank     := "DB_Wh_MOL".Tank[6]);
	
	"iDB_MOL_Tank_Log_7"(i_iRaw_AI  := "DB_IO_MAP".AI_MOL_Tank_7,
	                     i_rRaw_Siwa := 0.0,
	                     i_boRaw_DI  := "DB_IO_MAP".DI_MOL_Tank_7,
	                     io_Tank     := "DB_Wh_MOL".Tank[7]);
	
	"iDB_MOL_Tank_Log_8"(i_iRaw_AI  := "DB_IO_MAP".AI_MOL_Tank_8,
	                     i_rRaw_Siwa := 0.0,
	                     i_boRaw_DI  := "DB_IO_MAP".DI_MOL_Tank_8,
	                     io_Tank     := "DB_Wh_MOL".Tank[8]);
	
	"iDB_MOL_Tank_Log_9"(i_iRaw_AI  := "DB_IO_MAP".AI_MOL_Tank_9,
	                     i_rRaw_Siwa := 0.0,
	                     i_boRaw_DI  := "DB_IO_MAP".DI_MOL_Tank_9,
	                     io_Tank     := "DB_Wh_MOL".Tank[9]);
	
	"iDB_MOL_Tank_Log_10"(i_iRaw_AI  := "DB_IO_MAP".AI_MOL_Tank_10,
	                      i_rRaw_Siwa := 0.0,
	                      i_boRaw_DI  := "DB_IO_MAP".DI_MOL_Tank_10,
	                      io_Tank     := "DB_Wh_MOL".Tank[10]);
	
	"iDB_MOL_Tank_Log_11"(i_iRaw_AI  := "DB_IO_MAP".AI_MOL_Tank_11,
	                      i_rRaw_Siwa := 0.0,
	                      i_boRaw_DI  := "DB_IO_MAP".DI_MOL_Tank_11,
	                      io_Tank     := "DB_Wh_MOL".Tank[11]);
	
	"iDB_MOL_Tank_Log_12"(i_iRaw_AI  := "DB_IO_MAP".AI_MOL_Tank_12,
	                      i_rRaw_Siwa := 0.0,
	                      i_boRaw_DI  := "DB_IO_MAP".DI_MOL_Tank_12,
	                      io_Tank     := "DB_Wh_MOL".Tank[12]);
	
	// HMI маппинг
	FOR #temp_Ind := 1 TO 12 DO
	    "FC_Map_SmallTank_HMI"(i_Tank_Internal := "DB_Wh_MOL".Tank[#temp_Ind],
	                           io_HMI_Tank     := "DB_MAP".HMI_MOL_SmalTank[#temp_Ind]);
	END_FOR;
	
END_FUNCTION

FUNCTION "FC_Wh_POL_Mng" : Void
{ S7_Optimized_Access := 'FALSE' }
VERSION : 0.1
   VAR_TEMP 
      temp_Ind : Int;
   END_VAR


BEGIN
	// ---------------------------------------------------------------
	// Склад: Польский (POL) — 10 баков
	// Баки 1..3  — аналоговый уровень (AI)
	// Баки 4..10 — нет физических AI/DI (заглушки 0/FALSE для теста)
	// ---------------------------------------------------------------
	
	"iDB_POL_Tank_Log_1"(i_iRaw_AI  := "DB_IO_MAP".AI_POL_Tank_1,
	                     i_rRaw_Siwa := 0.0,
	                     i_boRaw_DI  := "DB_IO_MAP".DI_POL_Tank_1,
	                     io_Tank     := "DB_Wh_POL".Tank[1]);
	
	"iDB_POL_Tank_Log_2"(i_iRaw_AI  := "DB_IO_MAP".AI_POL_Tank_2,
	                     i_rRaw_Siwa := 0.0,
	                     i_boRaw_DI  := "DB_IO_MAP".DI_POL_Tank_2,
	                     io_Tank     := "DB_Wh_POL".Tank[2]);
	
	"iDB_POL_Tank_Log_3"(i_iRaw_AI  := "DB_IO_MAP".AI_POL_Tank_3,
	                     i_rRaw_Siwa := 0.0,
	                     i_boRaw_DI  := "DB_IO_MAP".DI_POL_Tank_3,
	                     io_Tank     := "DB_Wh_POL".Tank[3]);
	
	"iDB_POL_Tank_Log_4"(i_iRaw_AI  := "DB_IO_MAP".AI_POL_Tank_4,
	                     i_rRaw_Siwa := 0.0,
	                     i_boRaw_DI  := "DB_IO_MAP".DI_POL_Tank_4,
	                     io_Tank     := "DB_Wh_POL".Tank[4]);
	
	"iDB_POL_Tank_Log_5"(i_iRaw_AI  := "DB_IO_MAP".AI_POL_Tank_5,
	                     i_rRaw_Siwa := 0.0,
	                     i_boRaw_DI  := "DB_IO_MAP".DI_POL_Tank_5,
	                     io_Tank     := "DB_Wh_POL".Tank[5]);
	
	"iDB_POL_Tank_Log_6"(i_iRaw_AI  := "DB_IO_MAP".AI_POL_Tank_6,
	                     i_rRaw_Siwa := 0.0,
	                     i_boRaw_DI  := "DB_IO_MAP".DI_POL_Tank_6,
	                     io_Tank     := "DB_Wh_POL".Tank[6]);
	
	"iDB_POL_Tank_Log_7"(i_iRaw_AI  := "DB_IO_MAP".AI_POL_Tank_7,
	                     i_rRaw_Siwa := 0.0,
	                     i_boRaw_DI  := "DB_IO_MAP".DI_POL_Tank_7,
	                     io_Tank     := "DB_Wh_POL".Tank[7]);
	
	"iDB_POL_Tank_Log_8"(i_iRaw_AI  := "DB_IO_MAP".AI_POL_Tank_8,
	                     i_rRaw_Siwa := 0.0,
	                     i_boRaw_DI  := "DB_IO_MAP".DI_POL_Tank_8,
	                     io_Tank     := "DB_Wh_POL".Tank[8]);
	
	"iDB_POL_Tank_Log_9"(i_iRaw_AI  := "DB_IO_MAP".AI_POL_Tank_9,
	                     i_rRaw_Siwa := 0.0,
	                     i_boRaw_DI  := "DB_IO_MAP".DI_POL_Tank_9,
	                     io_Tank     := "DB_Wh_POL".Tank[9]);
	
	"iDB_POL_Tank_Log_10"(i_iRaw_AI  := "DB_IO_MAP".AI_POL_Tank_10,
	                      i_rRaw_Siwa := 0.0,
	                      i_boRaw_DI  := "DB_IO_MAP".DI_POL_Tank_10,
	                      io_Tank     := "DB_Wh_POL".Tank[10]);
	
	// HMI маппинг
	FOR #temp_Ind := 1 TO 10 DO
	    "FC_Map_SmallTank_HMI"(i_Tank_Internal := "DB_Wh_POL".Tank[#temp_Ind],
	                           io_HMI_Tank     := "DB_MAP".HMI_POL_SmalTank[#temp_Ind]);
	END_FOR;
	
END_FUNCTION

FUNCTION "FC_Wh_TRN_Mng" : Void
{ S7_Optimized_Access := 'FALSE' }
VERSION : 0.1
   VAR_TEMP 
      temp_Ind : Int;
   END_VAR


BEGIN
	"iDB_TRN_Tank_Log_1"(i_iRaw_AI:="DB_IO_MAP".AI_TRN_Tank_1,
	                     i_rRaw_Siwa:=0.0,
	                     i_boRaw_DI:="DB_IO_MAP".DI_TRN_Tank_1,
	                     io_Tank:="DB_Wh_TRN".Tank[1]);
	
	
	"iDB_TRN_Tank_Log_2"(i_iRaw_AI:=0,
	                     i_rRaw_Siwa:="DB_IO_MAP".AI_TRN_WTank_2,
	                     i_boRaw_DI:="DB_IO_MAP".DI_TRN_WTank_2,
	                     io_Tank:= "DB_Wh_TRN".Tank[2]);
	
	"iDB_TRN_Tank_Log_3"(i_iRaw_AI:=0,
	                     i_rRaw_Siwa:="DB_IO_MAP".AI_TRN_WTank_3,
	                     i_boRaw_DI:="DB_IO_MAP".DI_TRN_WTank_3,
	                     io_Tank:= "DB_Wh_TRN".Tank[3]);
	
	FOR #temp_Ind := 1 TO 3 DO
	    "FC_Map_SmallTank_HMI"(i_Tank_Internal := "DB_Wh_TRN".Tank[#temp_Ind],
	                           io_HMI_Tank := "DB_MAP".HMI_TRN_SmalTank[#temp_Ind]);
	END_FOR;
	
END_FUNCTION

FUNCTION "FC_ResetScaleCmd" : Void
{ S7_Optimized_Access := 'FALSE' }
VERSION : 0.1
   VAR_TEMP 
      tmp_Cmd : "UDT_SIWA_Cmd";
      tmp_Cmd_Raw AT tmp_Cmd : Array[0..3] of Byte;
   END_VAR


BEGIN
	// Зачищаем все 4 байта включая паддинг
	#tmp_Cmd_Raw[0] := 16#00;
	#tmp_Cmd_Raw[1] := 16#00;
	#tmp_Cmd_Raw[2] := 16#00;
	#tmp_Cmd_Raw[3] := 16#00;
	
	// Применяем ко всем слотам обоих модулей
	"DB_SCALE_CS_1".s_CMD1 := #tmp_Cmd;
	"DB_SCALE_CS_1".s_CMD2 := #tmp_Cmd;
	"DB_SCALE_CS_1".s_CMD3 := #tmp_Cmd;
	
	"DB_SCALE_CS_2".s_CMD1 := #tmp_Cmd;
	"DB_SCALE_CS_2".s_CMD2 := #tmp_Cmd;
	"DB_SCALE_CS_2".s_CMD3 := #tmp_Cmd;
END_FUNCTION

FUNCTION "FC_Scale_Map_Mng" : Void
{ S7_Optimized_Access := 'FALSE' }
VERSION : 0.1

BEGIN
	"iDB_Map_Siwarex_Core_1"(i_Scale_DB:="DB_Scale_CS_1",
	                         i_CycleTime_ms:=0,
	                         io_Core:="DB_MAP".Scale_CS_1);
	
	"iDB_Map_Siwarex_Core_2"(i_Scale_DB:="DB_Scale_CS_2",
	                         i_CycleTime_ms:=0,
	                         io_Core:="DB_MAP".Scale_CS_2);
	
END_FUNCTION

FUNCTION_BLOCK "FB_Sim_SawTooth_UpDown"
{ S7_Optimized_Access := 'FALSE' }
VERSION : 0.1
   VAR_INPUT 
      Enable : Bool;
      Speed : Real;
      Limit_High : Int := 27648;   // Верхний предел (по умолчанию максимум для аналогового входа Siemens)
      Limit_Low : Int := 0;   // Нижний предел
   END_VAR

   VAR_OUTPUT 
      Out_Raw : Int;
   END_VAR

   VAR_IN_OUT 
      Current_Val : Int;
   END_VAR

   VAR 
      Dir_Up : Bool := TRUE;   // Направление: TRUE = вверх, FALSE = вниз
   END_VAR

   VAR_TEMP 
      Increment : Int;
   END_VAR


BEGIN
	    // Если блок выключен, замораживаем текущее значение, сохраняем направление и выходим
	    IF NOT #Enable THEN
	        #Out_Raw := #Current_Val;
	        RETURN;
	    END_IF;
	    
	    // Рассчитываем шаг за цикл
	    #Increment := REAL_TO_INT(ABS(#Speed) * "getCycleTime"() / 1000.0);
	    
	    // Логика треугольного сигнала ("вверх-вниз")
	    IF #Dir_Up THEN
	        // Считаем вверх
	        #Current_Val := #Current_Val + #Increment;
	        IF #Current_Val >= #Limit_High THEN
	            #Current_Val := #Limit_High;
	            #Dir_Up := FALSE; // Меняем направление на "вниз"
	        END_IF;
	    ELSE
	        // Считаем вниз
	        #Current_Val := #Current_Val - #Increment;
	        IF #Current_Val <= #Limit_Low THEN
	            #Current_Val := #Limit_Low;
	            #Dir_Up := TRUE;  // Меняем направление на "вверх"
	        END_IF;
	    END_IF;
	    
	    // Обновляем выход
	    #Out_Raw := #Current_Val;
	    
END_FUNCTION_BLOCK

FUNCTION_BLOCK "CalculationVolume"
{ S7_Optimized_Access := 'FALSE' }
VERSION : 0.1
   VAR_INPUT 
      IW_Radius : Real;
      IW_ValueFromSensor : Real;
      IW_K_for_Tonnag : Real;
      IW_K_for_Level : Real;
   END_VAR

   VAR_OUTPUT 
      QW_Volume : Real;
      QW_Tonnag : Real;
      QW_RealLevel : Real;
   END_VAR

   VAR 
      sW_S : Real;
      sW_Volume : Real;
      sW_RealLevel : Real;
   END_VAR

   VAR CONSTANT 
      const_PI : Real := 3.14;
   END_VAR


BEGIN
	// Обрахування реального рівня
	#sW_RealLevel := #IW_ValueFromSensor / #IW_K_for_Level;
	
	// Обрахування площа перерізу 1 - для ємності,
	#sW_S := #const_PI * #IW_Radius * #IW_Radius;
	    
	// Volume = об*єм
	#sW_Volume := #sW_S * #sW_RealLevel;
	
	#QW_RealLevel := #sW_RealLevel; //реальний рівень
	#QW_Volume := #sW_Volume; //Присвоєння обрахованого обєму на вихід
	#QW_Tonnag := #sW_Volume * #IW_K_for_Tonnag; // обрахований обєм * Коефіцієнт
END_FUNCTION_BLOCK

FUNCTION_BLOCK "Analog_In_UDT"
{ S7_Optimized_Access := 'FALSE' }
AUTHOR : SimenCom
VERSION : 1.0
   VAR_INPUT 
      IB_Reset_PLC : Bool := false;
      IB_Total_Reset : Bool := false;
      IB_EnablePowerControl : Bool;
      IB_PowerControl : Bool;
      IW_HW_UpLevel : Int;
      IW_HW_LowLevel : Int;
      IW_Signal_from_Sensor : Int := 0;
   END_VAR

   VAR_OUTPUT 
      QW_STW : Array[0..15] of Bool;
      QDW_ScalledValue : Real;
      QB_HiHi_Fault : Bool;
      QB_Hi_Alarm : Bool;
      QB_Lo_Alarm : Bool;
      QB_LoLo_Fault : Bool;
      QB_Sensor_in_Zero : Bool;
   END_VAR

   VAR_IN_OUT 
      IUDT_Analog_In : "UDT_Analog_In";
   END_VAR

   VAR 
      Timer_TON_Filter {InstructionName := 'TON'; LibVersion := '1.0'} : TON;
      StB_Filter { ExternalAccessible := 'False'; ExternalVisible := 'False'; ExternalWritable := 'False'} : Bool;
      StDW_Sensor_After_Filter { ExternalAccessible := 'False'; ExternalVisible := 'False'; ExternalWritable := 'False'} : Real;
      StDW_Sensor_After_Scaling : Real;
      StB_HiHi : Bool;
      StB_Hi : Bool;
      StB_LoLo : Bool;
      StB_Lo : Bool;
      StB_HiHi_Q : Bool;
      StB_Hi_Q : Bool;
      StB_LoLo_Q : Bool;
      StB_Lo_Q : Bool;
      StB_PowerFault : Bool;
      Level_Control_HoLo : "Level_Control_HoLo";
      Smoothing_Instance : "Smoothing";
      Level_Control_HoLo_Instance : "Level_Control_HoLo";
   END_VAR

   VAR_TEMP 
      TmDW_Sensor_in_real : Real;
      TmB_Fault : Bool;
      TmDW_Sensor_After_DeadZone : Real;
      TmB_Reset_Bit : Bool;
      TmB_Sensor_In_Zero : Bool;
      TmDW_OutVal : Real;
   END_VAR


BEGIN
	// Help info 
	(*Біти в контрольних
	    словах:
	IW_CTW              
	0   -   Скиданя помилки -Кнопка-    SetBit
	1   -   Ввімкнути симуляцію -"Галочка"- SetBit
	2   -           
	3   -           
	4   -           
	5   -           
	6   -           
	7   -           
	8   -           
	9   -           
	10  -           
	11  -           
	12  -           
	13  -           
	14  -           
	15  -           
	    ************************************************************************
	    ************************************************************************
	QLW_STW     
	0   -   Все добре
	1   -   Активне попередження
	2   -   Загальна аварія
	3   -   Сигнал обриву давача 
	4   -   Досягнуто аварійного рівня (HiHi)
	5   -   Досягнуто рівня попередження (Hi)
	6   -   Опустилося нижче рівня попередження (Lo)
	7   -   Опустилося нижче аварійного рівня (LoLo)
	8   -   Симуляція ввімкнена
	9   -   Активне скидання помилок
	10  -   
	11  -   
	12  -   
	13  -   
	14  -   
	15  -   
	
	    ************************************************************************
	    ************************************************************************
	QDW_Message              
	0   -   Обрив лінії давача  -   Аварія
	1   -   Досягнуто аварійного рівня (HiHi)   -   Аварія
	2   -   Опустилося нижче аварійного рівня (LoLo)    -   Аварія
	3   -       -   
	4   -       -   
	5   -       -   
	6   -       -   
	7   -       -   
	8   -       -   
	9   -       -   
	10  -           
	11  -           
	12  -       -   
	13  -       -   
	14  -   Досягнуто рівня попередження (Hi)   -   Попередження
	15  -   Опустилося нижче рівня попередження (Lo)    -   Попередження
	16  -   Симуляція ввімкнена -   Подія
	17  -       -   
	18  -       -   
	19  -       -   
	20  -       -   
	
	*) 
	//Reset
	#TmB_Reset_Bit := #IB_Reset_PLC OR #IB_Total_Reset OR #IUDT_Analog_In.IW_CTW[0];
	
	//Логіка елементі живлення давача
	IF #IB_EnablePowerControl THEN
	    // #F_TRIG_PowerControl(CLK := #IB_PowerControl);
	    #StB_PowerFault := NOT #IB_PowerControl OR (#StB_PowerFault AND NOT #TmB_Reset_Bit);
	ELSE
	    #StB_PowerFault := false;
	END_IF;
	
	
	
	
	//Обрив давача
	IF  #IW_Signal_from_Sensor <= -32768 OR #IW_Signal_from_Sensor >= 32767 OR ((#StB_PowerFault OR NOT #IB_PowerControl) AND #IB_EnablePowerControl)  THEN
	    #TmB_Sensor_In_Zero := True;
	    #QB_Sensor_in_Zero := True;
	ELSE
	    #TmB_Sensor_In_Zero := False;
	    #QB_Sensor_in_Zero := False;
	END_IF;
	
	#TmDW_Sensor_in_real := INT_TO_REAL(#IW_Signal_from_Sensor);
	#IUDT_Analog_In.QW_HWValue := #IW_Signal_from_Sensor;
	
	// Згладжування сигналу . Масивне згладжування. Максимум 60 секунд
	#Smoothing_Instance(IDW_Input_Value := #TmDW_Sensor_in_real,
	                    IW_Time_Smoothing := #IUDT_Analog_In.IW_Time_Filter,
	                    IB_Gen_In := "tag_1",
	                    IW_Gen_Value := 200,
	                    QDW_Smoothing_Value => #StDW_Sensor_After_Filter);
	
	#TmDW_Sensor_in_real := 0;
	
	//Масштабування сигналу з множенням на коофіцієнт
	"Scaling_TSS"(In_Value := #StDW_Sensor_After_Filter,
	              In_Max := #IW_HW_UpLevel,
	              In_Min := #IW_HW_LowLevel,
	              Out_Max := #IUDT_Analog_In.IDW_UpLevel,
	              Out_Min := #IUDT_Analog_In.IDW_LowLevel,
	              Out_Value => #TmDW_OutVal,
	              Fault => #TmB_Fault,
	              Senser_In_Zero => #TmB_Fault);
	#StDW_Sensor_After_Scaling := #TmDW_OutVal * #IUDT_Analog_In.IDW_K_Mult;
	// "Мертва зона" сенсора
	IF #StDW_Sensor_After_Scaling >= #IUDT_Analog_In.IDW_DeadZone THEN
	#TmDW_Sensor_After_DeadZone := #StDW_Sensor_After_Scaling;
	ELSE
	    #TmDW_Sensor_After_DeadZone := 0;
	END_IF;
	
	
	// Обмеження симуляційного завдання
	IF #IUDT_Analog_In.IDW_Simulation_Value > #IUDT_Analog_In.IDW_UpLevel * #IUDT_Analog_In.IDW_K_Mult  THEN
	    #IUDT_Analog_In.IDW_Simulation_Value := #IUDT_Analog_In.IDW_UpLevel * #IUDT_Analog_In.IDW_K_Mult ;
	ELSIF #IUDT_Analog_In.IDW_Simulation_Value < #IUDT_Analog_In.IDW_LowLevel * #IUDT_Analog_In.IDW_K_Mult THEN
	    #IUDT_Analog_In.IDW_Simulation_Value := #IUDT_Analog_In.IDW_LowLevel * #IUDT_Analog_In.IDW_K_Mult ;
	END_IF;
	#TmDW_Sensor_in_real := 0;
	
	// Симуляція
	IF #IUDT_Analog_In.IW_CTW[0] THEN
	    #TmDW_Sensor_in_real := #IUDT_Analog_In.IDW_Simulation_Value;
	    #IUDT_Analog_In.QW_STW[8] := True;
	    
	ELSE
	    #TmDW_Sensor_in_real := #TmDW_Sensor_After_DeadZone;
	    #IUDT_Analog_In.QW_STW[8] := False;
	END_IF;
	
	//Блокування виходу при обриві
	IF NOT #TmB_Sensor_In_Zero OR #IUDT_Analog_In.IW_CTW[1] THEN
	    #QDW_ScalledValue := #TmDW_Sensor_in_real;
	    #IUDT_Analog_In.QDW_ScalledValue := #TmDW_Sensor_in_real;
	ELSE
	    #QDW_ScalledValue := 0.0;
	    #IUDT_Analog_In.QDW_ScalledValue := 0.0;
	    #TmDW_Sensor_in_real := 0.0;
	END_IF;
	
	// Логіка орпцювання аварійних повідомлень по сенсору
	// #IUDT_Analog_In.IBt_Block_ControlLevel.%X0 := true;
	// #IUDT_Analog_In.IBt_Block_ControlLevel.%X1 := true;
	// #IUDT_Analog_In.IBt_Block_ControlLevel.%X2 := true;
	// #IUDT_Analog_In.IBt_Block_ControlLevel.%X3 := true;
	#Level_Control_HoLo(IB_Enable_Func := NOT #TmB_Sensor_In_Zero,
	                    IDW_Actual_Value := #TmDW_Sensor_in_real,
	                    IDW_Set_HiHi := #IUDT_Analog_In.IDW_HiHi,
	                    IDW_Set_Hi := #IUDT_Analog_In.IDW_Hi,
	                    IDW_Set_LoLo := #IUDT_Analog_In.IDW_Lolo,
	                    IDW_Set_Lo := #IUDT_Analog_In.IDW_Lo,
	                    IW_Time_HiHi := #IUDT_Analog_In.IW_DelayON_HiHi,
	                    IW_Time_Hi := #IUDT_Analog_In.IW_DelayON_Hi,
	                    IW_Time_LoLo := #IUDT_Analog_In.IW_DelayON_LoLo,
	                    IW_Time_Lo := #IUDT_Analog_In.IW_DelayON_Lo);
	#StB_HiHi := (#StB_HiHi AND NOT #TmB_Reset_Bit)
	OR #IUDT_Analog_In.IBt_Enable_ControlLevel[0] AND #Level_Control_HoLo.QB_HiHi;
	#StB_HiHi_Q := (#StB_HiHi_Q AND NOT #TmB_Reset_Bit)
	OR #Level_Control_HoLo.QB_HiHi AND #IUDT_Analog_In.IBt_Block_ControlLevel[0];
	#QB_HiHi_Fault := #StB_HiHi_Q;
	
	#StB_Hi := #IUDT_Analog_In.IBt_Enable_ControlLevel[1] AND #Level_Control_HoLo.QB_Hi;
	#StB_Hi_Q := #Level_Control_HoLo.QB_Hi AND #IUDT_Analog_In.IBt_Block_ControlLevel[1];
	#QB_Hi_Alarm := #StB_Hi_Q;
	
	#StB_Lo := #IUDT_Analog_In.IBt_Enable_ControlLevel[2] AND #Level_Control_HoLo.QB_Lo;
	#StB_Lo_Q :=  #Level_Control_HoLo.QB_Lo AND #IUDT_Analog_In.IBt_Block_ControlLevel[2];
	#QB_Lo_Alarm := #StB_Lo_Q;
	
	#StB_LoLo := (#StB_LoLo AND NOT #TmB_Reset_Bit)
	OR #IUDT_Analog_In.IBt_Enable_ControlLevel[3] AND #Level_Control_HoLo.QB_LoLo;
	#StB_LoLo_Q := (#StB_LoLo_Q AND NOT #TmB_Reset_Bit)
	OR #Level_Control_HoLo.QB_LoLo AND #IUDT_Analog_In.IBt_Block_ControlLevel[3];
	#QB_LoLo_Fault := #StB_LoLo_Q;
	
	
	
	//IWCword
	#IUDT_Analog_In.IW_CTW[0] := False;
	
	//Word of State
	//Fault
	#IUDT_Analog_In.QW_STW[0] := #StB_HiHi OR #StB_LoLo OR #TmB_Sensor_In_Zero OR #StB_PowerFault;
	// Alarm
	#IUDT_Analog_In.QW_STW[1] := #StB_Hi OR #StB_Lo;
	// All OK
	#IUDT_Analog_In.QW_STW[2] := NOT #IUDT_Analog_In.QW_STW[0] AND NOT #IUDT_Analog_In.QW_STW[1];
	#IUDT_Analog_In.QW_STW[3] := #TmB_Sensor_In_Zero AND (( #IB_PowerControl AND #IB_EnablePowerControl) OR NOT #IB_EnablePowerControl );
	#IUDT_Analog_In.QW_STW[4] := #StB_HiHi;
	#IUDT_Analog_In.QW_STW[5] := #StB_Hi;
	#IUDT_Analog_In.QW_STW[6] := #StB_Lo;
	#IUDT_Analog_In.QW_STW[7] := #StB_LoLo;
	
	#IUDT_Analog_In.QW_STW[9] := #TmB_Reset_Bit;
	#IUDT_Analog_In.QW_STW[10] := #StB_PowerFault;
	#IUDT_Analog_In.QW_STW[11] := #IB_PowerControl;
	
	//Word of Alarm and fault
	#IUDT_Analog_In.QDW_Message[0] := #TmB_Sensor_In_Zero;
	#IUDT_Analog_In.QDW_Message[1] := #StB_HiHi;
	#IUDT_Analog_In.QDW_Message[2] := #StB_LoLo;
	#IUDT_Analog_In.QDW_Message[3] := #StB_PowerFault;
	
	#IUDT_Analog_In.QDW_Message[14] := #StB_Hi;
	#IUDT_Analog_In.QDW_Message[15] := #StB_Lo;
	
	#IUDT_Analog_In.QDW_Message[16] := #IUDT_Analog_In.QW_STW[8];
	
	#QW_STW := #IUDT_Analog_In.QW_STW;
	
	
END_FUNCTION_BLOCK

FUNCTION_BLOCK "Level_Control_HoLo"
{ S7_Optimized_Access := 'FALSE' }
VERSION : 0.1
   VAR_INPUT 
      IB_Enable_Func : Bool;
      IDW_Actual_Value : Real;
      IDW_Set_HiHi : Real;
      IDW_Set_Hi : Real;
      IDW_Set_LoLo : Real;
      IDW_Set_Lo : Real;
      IW_Time_HiHi : Int;
      IW_Time_Hi : Int;
      IW_Time_LoLo : Int;
      IW_Time_Lo : Int;
   END_VAR

   VAR_OUTPUT 
      QB_HiHi : Bool;
      QB_Hi : Bool;
      QB_LoLo : Bool;
      QB_Lo : Bool;
   END_VAR

   VAR 
      Timer_TON_HiHi {InstructionName := 'TON'; LibVersion := '1.0'} : TON;
      Timer_TON_Hi {InstructionName := 'TON'; LibVersion := '1.0'} : TON;
      Timer_TON_LoLo {InstructionName := 'TON'; LibVersion := '1.0'} : TON;
      Timer_TON_Lo {InstructionName := 'TON'; LibVersion := '1.0'} : TON;
   END_VAR

   VAR_TEMP 
      Tm_Time_HI : DInt;
      Tm_Time_Lo : DInt;
      Tm_Time_HIHI : DInt;
      Tm_Time_LOLO : DInt;
   END_VAR


BEGIN
	//Hi
	#Tm_Time_HI := INT_TO_DINT(#IW_Time_Hi);
	#Timer_TON_Hi(IN := #IDW_Actual_Value > #IDW_Set_Hi AND #IB_Enable_Func AND #IDW_Set_Hi <> 0,
	              PT := DINT_TO_TIME(#Tm_Time_HI * 1000),
	              
	              Q => #QB_Hi);
	
	//HiHi
	#Tm_Time_HIHI := INT_TO_DINT(#IW_Time_HiHi);
	#Timer_TON_HiHi(IN := #IDW_Actual_Value > #IDW_Set_HiHi AND #IB_Enable_Func AND #IDW_Set_HiHi <> 0,
	                PT := DINT_TO_TIME(#Tm_Time_HIHI * 1000),
	                Q => #QB_HiHi);
	//Lo
	#Tm_Time_Lo := INT_TO_DINT(#IW_Time_Lo);
	#Timer_TON_Lo(IN := #IDW_Actual_Value < #IDW_Set_Lo AND #IB_Enable_Func AND #IDW_Set_Lo <> 0,
	              PT := DINT_TO_TIME(#Tm_Time_Lo * 1000),
	              Q => #QB_Lo);
	//LoLo
	#Tm_Time_LOLO := INT_TO_DINT(#IW_Time_LoLo);
	#Timer_TON_LoLo(IN := #IDW_Actual_Value < #IDW_Set_LoLo AND #IB_Enable_Func AND #IDW_Set_LoLo <> 0,
	                PT := DINT_TO_TIME(#Tm_Time_LOLO * 1000),
	                Q => #QB_LoLo);
END_FUNCTION_BLOCK

FUNCTION_BLOCK "Smoothing"
{ S7_Optimized_Access := 'FALSE' }
VERSION : 0.1
   VAR_INPUT 
      IDW_Input_Value : Real;
      IW_Time_Smoothing : Int;
      IB_Gen_In : Bool;
      IW_Gen_Value : DInt;
   END_VAR

   VAR_OUTPUT 
      QDW_Smoothing_Value : Real;
   END_VAR

   VAR 
      Value_array : Array[0..100] of Real;
      St_PointArray : Int;
      St_Counter : Int;
      St_Counter_Shift : Int;
      St_Counter_Summ : Int;
      St_Summ_Arr : Real;
   END_VAR

   VAR_TEMP 
      Temp_UDint : DInt;
   END_VAR


BEGIN
	#Temp_UDint := #IW_Time_Smoothing;
	IF #IW_Time_Smoothing>0 THEN
	        
	    #St_PointArray := (DINT_TO_INT((#Temp_UDint * 100) / #IW_Gen_Value));
	    IF #St_PointArray>100
	    THEN
	        #St_PointArray := 100;
	    END_IF;
	    
	    //#R_TRIG_Instance(CLK:=#IB_Gen_In);
	    
	    IF #IB_Gen_In THEN
	        
	        #St_Summ_Arr := 0;
	        FOR #St_Counter_Shift := #St_PointArray  TO 2 BY -1 DO
	            #Value_array[#St_Counter_Shift] := #Value_array[#St_Counter_Shift - 1];
	        END_FOR;
	        #Value_array[1] := #IDW_Input_Value;
	        //Обмеження лічильника
	        IF #St_Counter<#St_PointArray THEN
	            #St_Counter := #St_Counter + 1;
	        ELSE
	            #St_Counter := #St_PointArray;
	        END_IF;
	        //Сумування масиву
	        FOR #St_Counter_Summ := 1 TO #St_Counter DO
	            #St_Summ_Arr := #St_Summ_Arr + #Value_array[#St_Counter_Summ];
	        END_FOR;
	        //Усереднене значення масиву
	        #QDW_Smoothing_Value := #St_Summ_Arr / (#St_Counter);
	    END_IF;
	    
	ELSE
	#QDW_Smoothing_Value := #IDW_Input_Value;
	#St_Counter := 0;
	END_IF;
	
	
	
	
END_FUNCTION_BLOCK

FUNCTION "Scaling_TSS" : Void
{ S7_Optimized_Access := 'FALSE' }
VERSION : 0.1
   VAR_INPUT 
      In_Value : Real;
      In_Max : Real;
      In_Min : Real;
      Out_Max : Real;
      Out_Min : Real;
   END_VAR

   VAR_OUTPUT 
      Out_Value : Real;
      Fault : Bool;
      Senser_In_Zero : Bool;
   END_VAR

   VAR_TEMP 
      Diap_In : Real;
      Diap_Out : Real;
      In_prop : Real;
      Out_prop_1 : Real;
      Value_Out : Real;
      Value_IN : Real;
      Temp_Sensor_In_Zero : Bool;
   END_VAR


BEGIN
	#Diap_In := #In_Max - #In_Min;
	#Diap_Out := #Out_Max - #Out_Min;
	#Value_IN := #In_Value - #In_Min;
	IF #In_Max < #In_Min                                   //Перевірка чи максимальні значення не менші мінімальних
	    OR (#Out_Max < #Out_Min)                         //якщо так то помилка 
	THEN
	    #Fault := true;
	    
	ELSE
	    //Перевірка чи апаратне значення не за доступними межами; якщо так то датчик в нулі
	    // IF #In_Value = 32768
	    //     OR (#In_Value = -32768)
	    // THEN
	    //     #Senser_In_Zero := true;
	    //     #Temp_Sensor_In_Zero := true;
	    //     #Out_Value := 0;
	    // ELSE
	    //     #Senser_In_Zero := false;
	    //     #Temp_Sensor_In_Zero := false;
	    // END_IF;
	    
	    #Fault := false;
	    #In_prop := (#Value_IN * 100) / #Diap_In;                    //Вхід в процентах
	    #Out_prop_1 := (#Diap_Out * 1) / 100;                       //1 процент від шкали виходу
	    #Value_Out := #In_prop * #Out_prop_1;                       //Вихід в процентах    
	    
	    IF #In_Value > #In_Max
	        // AND NOT (#Temp_Sensor_In_Zero)
	    THEN
	        #Out_Value := #Out_Max;
	    ELSIF #In_Value < #In_Min
	        // AND NOT (#Temp_Sensor_In_Zero)
	    THEN
	        #Out_Value := #Out_Min;
	    ELSIF #In_Value >= #In_Min AND #In_Value <= #In_Max
	        // AND NOT #Temp_Sensor_In_Zero
	    THEN
	        #Out_Value := #Out_Min + #Value_Out;
	    END_IF;
	    
	    
	END_IF;
	
	
	
	
	
END_FUNCTION
